"F0ERPLA"	Q 600.4	BOOL	// [F0IM1.F0S11]: F0: EV RECUO PILOTO A
"F0ERSRB"	Q 600.5	BOOL	// [F0IM1.F0S11]: F0: EV RECUO SERRAGE B
"F0IM_F0S11_R1"	Q 600.6	BOOL	// [F0IM1.F0S11]: RESERVA
"F0ERSRD"	Q 600.7	BOOL	// [F0IM1.F0S11]: F0: EV RECUO SERRAGE D
"F0ERRCE"	Q 601.0	BOOL	// [F0IM1.F0S12]: F0: EV RECUO RETACAGE E
"F0EACAF"	Q 601.1	BOOL	// [F0IM1.F0S12]: F0: EV AVANÇO CARRO F
"F0EARCF1"	Q 601.2	BOOL	// [F0IM1.F0S12]: F0: EV AVANÇO RETACAGE F1
"F0IM_F0S12_R1"	Q 601.3	BOOL	// [F0IM1.F0S12]: RESERVA
"F0EARCE"	Q 601.4	BOOL	// [F0IM1.F0S12]: F0: EV AVANÇO RETACAGE E
"F0ERCAF"	Q 601.5	BOOL	// [F0IM1.F0S12]: F0: EV RECUO CARRO F
"F0IM_F0S12_R2"	Q 601.6	BOOL	// [F0IM1.F0S12]: RESERVA
"F0IM_F0S12_R3"	Q 601.7	BOOL	// [F0IM1.F0S12]: RESERVA
"G0EAPLA"	Q 620.0	BOOL	// [G0IM1.G0S11]: G0: EV AVANÇO PILOTO A
"G0EASRB"	Q 620.1	BOOL	// [G0IM1.G0S11]: G0: EV AVANÇO SERRAGE B
"G0IM_G0S13_R1"	Q 620.2	BOOL	// [G0IM1.G0S11]: RESERVA
"G0IM_G0S13_R2"	Q 620.3	BOOL	// [G0IM1.G0S11]: RESERVA
"G0ERPLA"	Q 620.4	BOOL	// [G0IM1.G0S11]: G0: EV RECUO PILOTO A
"G0ERSRB"	Q 620.5	BOOL	// [G0IM1.G0S11]: G0: EV RECUO SERRAGE B
"G0IM_G0S13_R3"	Q 620.6	BOOL	// [G0IM1.G0S11]: RESERVA
"G0IM_G0S13_R4"	Q 620.7	BOOL	// [G0IM1.G0S11]: RESERVA
"RESERVA-"	Q 640.7	BOOL	// [H0IM1.H0S11]: H0: RESERVA
"K0EASR1"	Q 650.0	BOOL	// [K0TDS1] K0: EV AVANCE SR1
"K0ERSR1"	Q 650.1	BOOL	// [K0TDS1] K0: EV RETROCESO SR1
"K0EASR2"	Q 650.2	BOOL	// [K0TDS1] K0: EV AVANCE SR2
"K0ERSR2"	Q 650.3	BOOL	// [K0TDS1] K0: EV RETROCESO SR2
"K0S11_RESERVA1"	Q 650.4	BOOL
"K0S11_RESERVA2"	Q 650.5	BOOL
"K0EASR3"	Q 650.6	BOOL	// [K0TDS1] K0: EV AVANCE SR3
"K0ERSR3"	Q 650.7	BOOL	// [K0TDS1] K0: EV RETROCESO SR3
"K0_VVAL"	Q 656.0	BOOL	// [K0A2] Habilitacion de 24V Valvulas CPX K0TDS1
"K0EVCPX"	Q 656.1	BOOL	// [K0A2] ELECTROVÁLVULA CPX K0TDS1
"Z2RCM"	Q 800.7	BOOL	// [Z2ZB.M05]: Z2 GROUND CONTROL RELAY
"Z2RSC1"	Q 815.0	BOOL	// [Z2ZB.M09]: RELAY SAFETY COMMON 1 (AU)
"Z2RES"	Q 815.1	BOOL	// [Z2ZB.M09]: RELAY SAFETY COMMON 2 (ES)
"Z2RFZ"	Q 815.2	BOOL	// [Z2ZB.M09]: RELAY SAFETY COMMON 3 (RFZ)
"Z2RSC4"	Q 815.3	BOOL	// [Z2ZB.M09]: RELAY SAFETY COMMON 4 (SC4)
"B1OP1VAT"	Q 821.0	BOOL	// B1 Lampara autorizacion de trabajo
"B1OP1VIT"	Q 821.1	BOOL	// B1 Lampara de prohibicion de trabajo
"B1OP1VDF"	Q 821.2	BOOL	// B1 Lampara de defecto
"B0RFRO1"	Q 841.0	BOOL	// [B0SB.M11]: B0 SAFETY COMMON 3 (FRO1)
"B0RFRO2"	Q 841.1	BOOL	// [B0SB.M11]: B0 SAFETY COMMON 4 (FRO2)
"B0RFRO3"	Q 841.2	BOOL	// [B0SB.M11]: B0 SAFETY COMMON 5 (FRO3)
"C1OP1VAT"	Q 851.0	BOOL	// C1 Lampara autorizacion de trabajo
"C1OP1VIT"	Q 851.1	BOOL	// C1 Lampara de prohibicion de trabajo
"C1OP1VDF"	Q 851.2	BOOL	// C1 Lampara de defecto
"C0RFRO1"	Q 871.0	BOOL	// [C0SB.M11]: C0 SAFETY COMMON 3 (C0SOP)
"C0RFRO2"	Q 871.1	BOOL	// [C0SB.M11]: C0 SAFETY COMMON 4 (C0)
"C0RFRO3"	Q 871.2	BOOL	// [C0SB.M11]: C0 SAFETY COMMON 5 (C0)
"E1OP1VAT"	Q 881.0	BOOL	// E1 Lampara autorizacion de trabajo
"E1OP1VIT"	Q 881.1	BOOL	// E1 Lampara de prohibicion de trabajo
"E1OP1VDF"	Q 881.2	BOOL	// E1 Lampara de defecto
"E2OP2VAT"	Q 881.5	BOOL
"E2OP2VIT"	Q 881.6	BOOL
"E0RFRO1"	Q 901.0	BOOL	// [E0SB.M11]: E0 SAFETY COMMON 3 ( E0SOP)
"E0RFRO2"	Q 901.1	BOOL	// [E0SB.M11]: E0 SAFETY COMMON 4 ( E0)
"E0RFRO3"	Q 901.2	BOOL	// [E0SB.M11]: E0 SAFETY COMMON 5 ( E0)
"G1OP1VAT"	Q 911.0	BOOL	// B1 Lampara autorizacion de trabajo
"G1OP1VIT"	Q 911.1	BOOL	// B1 Lampara de prohibicion de trabajo
"G1OP1VDF"	Q 911.2	BOOL	// B1 Lampara de defecto
"G0RFRO1"	Q 931.0	BOOL	// [G0SB.M11]: G0 SAFETY COMMON 3 (G0SOP)
"G0RFRO2"	Q 931.1	BOOL	// [G0SB.M11]: G0 SAFETY COMMON 4 (G0)
"G0RFRO3"	Q 931.2	BOOL	// [G0SB.M11]: G0 SAFETY COMMON 5 (G0)
"J1OP1VAT"	Q 940.0	BOOL	// J1 Lampara autorizacion de trabajo
"J1OP1VIT"	Q 940.1	BOOL	// J1 Lampara de prohibicion de trabajo
"J1OP1VDF"	Q 940.2	BOOL	// J1 Lampara de defecto
"B0EAPL1"	Q 950.0	BOOL	// [B0DTS1]: B0: EV AVANCE PL1
"B0ERPL1"	Q 950.1	BOOL	// [B0DTS1]: B0: EV RETROCESO PL1
"B0EASR2"	Q 950.2	BOOL	// [B0DTS1]: B0: EV AVANCE SR2
"B0ERSR2"	Q 950.3	BOOL	// [B0DTS1]: B0: EV RETROCESO SR2
"B0EASR3"	Q 950.4	BOOL	// [B0DTS1]: B0: EV AVANCE SR3
"B0ERSR3"	Q 950.5	BOOL	// [B0DTS1]: B0: EV RETROCESO SR3
"C0EAPL1"	Q 960.0	BOOL	// [C0DTS1]: C0: EV AVANCE PL1
"C0ERPL1"	Q 960.1	BOOL	// [C0DTS1]: C0: EV RETROCESO PL1
"C0EASR2"	Q 961.2	BOOL	// [C0DTS1]: C0: EV AVANCE SR2
"C0ERSR2"	Q 961.3	BOOL	// [C0DTS1]: C0: EV RETROCESO SR2
"C0EASR3"	Q 961.4	BOOL	// [C0DTS1]: C0: EV AVANCE SR3
"C0ERSR3"	Q 961.5	BOOL	// [C0DTS1]: C0: EV RETROCESO SR3
"E0EASR1"	Q 1040.0	BOOL	// [E0TDS1]: E0: EV AVANCE SR1
"E0ERSR1"	Q 1040.1	BOOL	// [E0TDS1]: E0: EV RETROCESO SR1
"E0EASR2"	Q 1040.2	BOOL	// [E0TDS1]: E0: EV AVANCE SR2
"E0ERSR2"	Q 1040.3	BOOL	// [E0TDS1]: E0: EV RETROCESO SR2
"E0EASR3"	Q 1040.4	BOOL	// [E0TDS1]: E0: EV AVANCE SR3
"E0ERSR3"	Q 1040.5	BOOL	// [E0TDS1]: E0: EV RETROCESO SR3
"E0EAVU4"	Q 1040.6	BOOL	// [E0TDS1]: E0: EV AVANCE VU4
"E0ERVU4"	Q 1040.7	BOOL	// [E0TDS1]: E0: EV RETROCESO VU4
"E0EAVU5"	Q 1041.0	BOOL	// [E0TDS1]: E0: EV AVANCE VU5
"E0ERVU5"	Q 1041.1	BOOL	// [E0TDS1]: E0: EV RETROCESO VU5
"E0EASR6"	Q 1041.2	BOOL	// [E0TDS1]: E0: EV AVANCE SR6
"E0ERSR6"	Q 1041.3	BOOL	// [E0TDS1]: E0: EV RETROCESO SR6
"G0EASR1"	Q 1060.0	BOOL	// [G0TDS1]: G0: EV AVANCE SR1
"G0ERSR1"	Q 1060.1	BOOL	// [G0TDS1]: G0: EV RETROCESO SR1
"G0EASR2"	Q 1060.2	BOOL	// [G0TDS1]: G0: EV AVANCE SR2
"G0ERSR2"	Q 1060.3	BOOL	// [G0TDS1]: G0: EV RETROCESO SR2
"G0EASR3"	Q 1060.4	BOOL	// [G0TDS1]: G0: EV AVANCE SR3
"G0ERSR3"	Q 1060.5	BOOL	// [G0TDS1]: G0: EV RETROCESO SR3
"L1VROC"	Q 1070.0	BOOL	// L1: LED BOTON RETORNO A ORIGEN
"L1VIT"	Q 1070.2	BOOL	// L1: LAMPARA DE PROHIBICION DE TRABAJO
"L1VDF"	Q 1070.3	BOOL	// L1: LAMPARA DE DEFECTO
"L1VAT"	Q 1070.4	BOOL	// L1: LAMPARA DE PROHIBICION DE TRABAJO
"L0EAPS1"	Q 1071.0	BOOL	// L0: Electrovalvula de avance PIN SHIFT 1
"L0ERPS1"	Q 1071.1	BOOL	// L0: Electrovalvula de retroceso PIN SHIFT 1
"L0EASR1"	Q 1071.2	BOOL	// L0: Electrovalvula de avance CLAMP 1
"L0ERSR1"	Q 1071.3	BOOL	// L0: Electrovalvula de retroceso CLAMP 1
"L0EASR2"	Q 1071.4	BOOL	// L0: Electrovalvula de avance CLAMP 2
"L0ERSR2"	Q 1071.5	BOOL	// L0: Electrovalvula de retroceso CLAMP 2
"L0EASR3"	Q 1071.6	BOOL	// L0: Electrovalvula de avance CLAMP 3
"L0ERSR3"	Q 1071.7	BOOL	// L0: Electrovalvula de retroceso CLAMP 3
"L0EAVU1"	Q 1072.0	BOOL	// L0: Electrovalvula de avance EJECTOR 1
"L0ERVU1"	Q 1072.1	BOOL	// L0: Electrovalvula de retroceso EJECTOR 1
"L0EAVU2"	Q 1072.2	BOOL	// L0: Electrovalvula de avance PINGYI 1
"L0ERVU2"	Q 1072.3	BOOL	// L0: Electrovalvula de retroceso PINGYI 1
"L0EASR4"	Q 1072.4	BOOL	// L0: ELECTROVALVULA DE AVANCE MOV SR4 (DETECTOR DPP15)
"L0ERSR4"	Q 1072.5	BOOL	// L0: ELECTROVALVULA DE AVANCE MOV SR4 (DETECTOR DPP15)
"FDIS_90_8_AckCan"	Q 1080.0	BOOL	// FESTO DI-Safe error de canal 90 - 8 L0
"FDIS_90_8_Pass"	Q 1080.1	BOOL	// FESTO DI-Safe 90 - 8 1 PASSIVATION PAR CANAL / 0 - PASSIVATION PAR MODULE
"L0SOP"	Q 1087.0	BOOL
"L024SV"	Q 1087.1	BOOL	// L0 24V SUPPLY FOR SOFSTART VALVE
"M1VROC"	Q 1100.0	BOOL	// M1: LAMPARA DE RETORNO AL ORIGEN
"M1VIT"	Q 1100.2	BOOL	// M1: LAMPARA DE PROHIBICION DE TRABAJO
"M1VDF"	Q 1100.3	BOOL	// M1: LAMPARA DE DEFECTO
"M1VAT"	Q 1100.4	BOOL	// M1: LAMPARA DE PERMISO DE TRABAJO
"FDIS_100_5_AckCan"	Q 1104.0	BOOL	// FESTO DI-Safe ERROR DE CANAL M0
"FDIS_100_5_Pass"	Q 1104.1	BOOL	// FESTO DI-Safe 1 - passivation par canal / 0 - passivation par module
"M0SOP"	Q 1111.0	BOOL
"M024SV"	Q 1111.1	BOOL	// M0 24V SUPPLY FOR SOFSTART VALVE
"M0EASR1"	Q 1117.0	BOOL	// M0: Electrovalvula avance HAND CLAMP 1
"M0ERSR1"	Q 1117.1	BOOL	// M0: Electrovalvula retroceso HAND CLAMP 1
"M0EASR2"	Q 1117.2	BOOL	// M0: Electrovalvula avance CLAMP 1
"M0ERSR2"	Q 1117.3	BOOL	// M0: Electrovalvula retroceso CLAMP 1
"M0EAVU1"	Q 1117.4	BOOL	// M0: Electrovalvula avance EJECTOR 1
"M0ERVU1"	Q 1117.5	BOOL	// M0: Electrovalvula retroceso EJECTOR 1
"N0EAPLC"	Q 1150.4	BOOL
"N0ERPLC"	Q 1150.5	BOOL
"N0EASRD"	Q 1150.6	BOOL
"N0ERSRD"	Q 1150.7	BOOL
"N0EASRE"	Q 1151.0	BOOL
"N0ERSRE"	Q 1151.1	BOOL
"N0EASRF"	Q 1151.2	BOOL
"N0ERSRF"	Q 1151.3	BOOL
"N0EACLH"	Q 1151.6	BOOL
"N0ERCLH"	Q 1151.7	BOOL
"N0EASRJ"	Q 1152.0	BOOL
"N0ERSRJ"	Q 1152.1	BOOL
"N0EACLK"	Q 1152.2	BOOL
"N0ERCLK"	Q 1152.3	BOOL
"N0EBLK"	Q 1152.4	BOOL	// ElectroValvula Bloqueti Cilindro K
"N1VDF"	Q 1155.0	BOOL	// N1: LAMPARA DE DEFECTO
"N1VAT"	Q 1155.1	BOOL	// N1: LAMPARA DE PERMISO DE TRABAJO
"N1VIT"	Q 1155.3	BOOL	// N1: LAMPARA DE PROHIBICION DE TRABAJO
"N0EAPLA"	Q 1156.0	BOOL
"N0ERPLA"	Q 1156.1	BOOL
"N0EACLB"	Q 1156.2	BOOL
"N0ERCLB"	Q 1156.3	BOOL
"N0EACLG"	Q 1156.4	BOOL
"N0ERCLG"	Q 1156.5	BOOL
"FDIS_110_5_AckCan"	Q 1158.0	BOOL	// FESTO DI-Safe ERROR DE CANAL M0
"FDIS_110_5_Pass"	Q 1158.1	BOOL	// FESTO DI-Safe 1 - passivation par canal / 0 - passivation par modul
"N0SOP"	Q 1165.0	BOOL	// N0IM1: COMUN SEGURIDAD OPERADO
"N0EVAIR"	Q 1165.1	BOOL	// N0 ELECTROVALVULA DE AIRE GENERAL
"FDIS_90_8_M"	QW 1081	INT	// FESTO DI-Safe 90-8 MODE L0
"FDIS_100_5_M"	QW 1105	INT	// FESTO DI-Safe 100 - 5 MODE
"FDIS_110_5_M"	QW 1159	INT	// FESTO DI-Safe 110 - 5 MODE
"TP"	SFB 3	SFB 3	// GENERATE A PULSE
"TON"	SFB 4	SFB 4	// GENERATE AN ON DELAY
"TOF"	SFB 5	SFB 5	// GENERATE AN OFF DELAY
"RDREC"	SFB 52	SFB 52	// READ A PROCESS DATA RECORD
"WRREC"	SFB 53	SFB 53	// WRITE A PROCESS DATA RECORD
"RALRM"	SFB 54	SFB 54	// Receive Alarm Data
"SET_CLK"	SFC 0	SFC 0	// SET SYSTEM CLOCK
"READ_CLK"	SFC 1	SFC 1	// READ SYSTEM CLOCK
"RD_SINFO"	SFC 6	SFC 6	// READ OB START INFORMATION
"D_ACT_DP"	SFC 12	SFC 12	// DEACTIVATING AND ACTIVATING DP SLAVES
"DPRD_DAT"	SFC 14	SFC 14	// READ CONSISTENT DATA OF A STANDARD DP SLAVE
"DPWR_DAT"	SFC 15	SFC 15	// WRITE CONSISTENT DATA TO A STANDARD DP SLAVE
"BLKMOV"	SFC 20	SFC 20	// COPY VARIABLES
"FILL"	SFC 21	SFC 21	// INITIALIZE A MEMORY AREA
"TEST_DB"	SFC 24	SFC 24	// TEST DATA BLOCK
"DIS_AIRT"	SFC 41	SFC 41	// DELAY THE HIGHER PRIORITY INTERRUPTS AND ASYNCHRONOUS ERRORS
"EN_AIRT"	SFC 42	SFC 42	// ENABLE HIGHER PRIORITY INTERRUPTS AND ASYNCHRONOUS ERRORS
"STP"	SFC 46	SFC 46	// CHANGE THE CPU TO STOP
"RDSYSST"	SFC 51	SFC 51	// READ A SYSTEM STATUS LIST OR PARTIAL LIST
"WR_REC"	SFC 58	SFC 58	// WRITE DATA RECORD
"RD_REC"	SFC 59	SFC 59	// READ A DATA RECORD
"TIME_TCK"	SFC 64	SFC 64	// READ THE SYSTEM TIME
"GEO_LOG"	SFC 70	SFC 70	// DETERMINE LOGICAL ADDRESS
"READ_DBL"	SFC 83	SFC 83	// READ DATA BLOCK OUT OF LOAD MEMORY
"WRIT_DBL"	SFC 84	SFC 84	// WRITE DATA BLOCK IN LOAD MEMORY
"DEL_SI"	SFC 106	SFC 106	// Deleting Dynamically Assigned System Instances
"ALARM_DQ"	SFC 107	SFC 107	// Creating Acknowledgeable Block-related Message
"ALARM_D"	SFC 108	SFC 108	// Creating Acknowledged Block-related Message
"LIEN_SEC"	UDT 1507	UDT 1507	// TABLE COMMUNE AUX BF_ZONE_PORTE1, BF_ZONE_RSEC1, BF_ZONE_MODE_IHM, BF_ZONE_AIR
"MOT_FONC_DPL"	UDT 1866	UDT 1866
"LIEN_PUP"	UDT 1988	UDT 1988	// Gestion des Modes et des pupitres de cde manu de la  zone (BF_ZONE_MODE_IHM)
"LIEN_ILOT"	UDT 2004	UDT 2004	// INFO CONTROL LINKED TO THE FACILITY (BF_ILOT)
"MOT_FONC_MP"	UDT 2041	UDT 2041	// INFO CONTROL OF A MOVEMENT (BF_MOUVMP1)
"MOT_FONC"	UDT 2042	UDT 2042	// INFO D'UN MOUVEMENT (BF_MOUV2P1,BF_MVSE2P1, BF_RB_COD_PREH_API)
"VAT_SIPTOL"	VAT 1	
"VAT_TALOA0"	VAT 2	
"VAT_BASE DE DADOS"	VAT 3	
"Z1T_TEMPOS"	VAT 4	
"Z2T_TEMPOS"	VAT 5	
"VAT_6"	VAT 6	
"acompanhamento zona 8"	VAT 7		// teste tucker
"TOMAS"	VAT 8	
"W0"	VAT 9	
"VAT_Z1_BOT_EMER"	VAT 10	
"VAT_Z2_BOT_EMER"	VAT 11		// BOTAO_DE_EMERGENCIA
"VAT_Z1_VALIDAÇÃO"	VAT 12	
"VAT_CDIV_2"	VAT 13	
"VAT_Z2_VALIDAÇÃO"	VAT 14	
"ELEV_CARREGAMENTO"	VAT 15	
"ELEV_DESCARREGAMENTO"	VAT 16	
"VAT_17"	VAT 17	
"TESTE_MODO_DEGR"	VAT 18	
"Z2_SIPTOL"	VAT 19	
"mostrar IIT"	VAT 20	
"tab_iit_2"	VAT 21	
"VAT_22"	VAT 22	
"afficher"	VAT 23	
"VAT_24"	VAT 24	
"SIPTOL_X52_X67_X60"	VAT 25	
"Z3_SIPTOL"	VAT 26		// VAT SIPTOL ZONA 3
"VAT_IIT"	VAT 27	
"VAT_Z1T"	VAT 28	
"SMP"	VAT 29	
"def_qbad"	VAT 30	
END_SYMBOL_TABLE

SYMBOL_TABLE
"CC1"	C 1	COUNTER	// Contador Cabeçote 1
"CC2"	C 2	COUNTER	// Contador Cabeçote 2
"CC3"	C 3	COUNTER	// Contador Cabeçote 3
"CT_M6_FAG0014"	C 4	COUNTER	// Contador de tucker pistola 1 do DCE FAG0014
"CT_M6_FAG0039"	C 5	COUNTER	// Contador de tucker pistola 3 do DCE FAG0039
"CT_P1M6_RF60"	C 6	COUNTER	// CONTADOR PISTOLA 1 M6 RF60
"CT_P2M6_RF60"	C 7	COUNTER	// CONTADOR PISTOLA 2 M6 RF60
"I01"	DB 1	FB 1	// FACILITY: INSTANCE DB (FB1)
"I02"	DB 2	FB 2	// FACILITY: INSTANCE DB FOR MMC CONTROL (FB2)
"I03"	DB 3	FB 3	// FACILITY: INSTANCE DB FOR MOP/LOP
"I04"	DB 4	FB 4
"CDIV"	DB 69	DB 69	// FACILITY: DIVERSITIES CODES TABLE / TABLE CODES DIVERSITES
"SFM_DB"	DB 75	FB 20	// FACILITY: DB FAILURE MESSAGE (SFM_FB) LINK WITH PROFINET CONTROL
"SFM_GLOBAL_DB"	DB 76	DB 76	// DIAGNOSTIC BLOCK FOR THE SIGNALISATION OF THE SYSTEM ERRORS
"SFM_PN"	DB 77	DB 77	// PROFINET DIAGNOSTIC FUNCTION EDITING DB FOR IHMP
"SIP1"	DB 89	DB 89	// SIPTOL EXCHANGES DATAS / TABLE D'ECHANGES SIPTOL
"PILE"	DB 90	DB 90	// FACILITY: FIFO STORAGE / PILE DE STOCKAGE
"CAB"	DB 91	DB 91	// L0: BARCODE READER DB / DB LECTEUR CODE BARRE
"IDENT"	DB 93	DB 93	// RFID DATAS / IDENTIFIANT DYNAMIQUE
"IBD"	DB 95	DB 95	// FACILITY: DATA BASE DB / DB BASE DE DONNEE
"IIT"	DB 96	DB 96	// FACILITY: PART TABLE / DB TABLE PIECE
"IG"	DB 99	DB 99	// FACILITY: GLOBAL DB / DB GLOBAL
"Z1"	DB 100	FB 100	// ZONE 1: INSTANCE DB
"Z1A0"	DB 110	FB 110	// A0 MONTAGE INSTANCE DATA BLOC / BLOC DE DONNEES INSTANCE A0 MONTAGE
"Z1A1"	DB 111	FB 111	// A1 OP_BIMA INSTANCE DATA BLOC / BLOC DE DONNEES INSTANCE A1 OP_BIMA
"Z1A2"	DB 112	FB 112	// A2 OP_BIMA INSTANCE DATA BLOC / BLOC DE DONNEES INSTANCE A2 OP_BIMA
"Z1A0L"	DB 114	FB 114	// A0 LANCEMENT INSTANCE DATA BLOC / BLOC DE DONNEES INSTANCE A0 LANCEMENT
"Z1D0"	DB 140	FB 140	// D0 MONTAGE INSTANCE DATA BLOC / BLOC DE DONNEES INSTANCE D0 MONTAGE
"Z1D1"	DB 141	FB 141	// D1 OP_BIMA INSTANCE DATA BLOC / BLOC DE DONNEES INSTANCE D1 OP_BIMA
"Z1D2"	DB 142	FB 142	// D2 OP_BIMA INSTANCE DATA BLOC / BLOC DE DONNEES INSTANCE D2 OP_BIMA
"Z1F0"	DB 150	FB 150	// F0 MONTAGE INSTANCE DATA BLOC / BLOC DE DONNEES INSTANCE F0 MONTAGE
"Z1F1"	DB 151	FB 151	// F1 OP_BIMA INSTANCE DATA BLOC / BLOC DE DONNEES INSTANCE F1 OP_BIMA
"Z1F2"	DB 152	FB 152	// F2 OP_BIMA INSTANCE DATA BLOC / BLOC DE DONNEES INSTANCE F2 OP_BIMA
"Z1F3"	DB 153	FB 253	// F3 OP_BIMA INSTANCE DATA BLOC / BLOC DE DONNEES INSTANCE F3 OP_BIMA
"Z1N0"	DB 160	FB 160
"Z1N1"	DB 161	FB 161
"Z1K0"	DB 170	FB 170
"Z1K1"	DB 171	FB 171
"Z1T"	DB 198	DB 198	// ZONE 1: REFERENCE TIME FOR MOVEMENTS
"Z1G"	DB 199	DB 199	// ZONE 1: GLOBAL DB
"Z2"	DB 200	FB 200	// ZONE 2: INSTANCE DB
"Z2B0"	DB 210	FB 210
"Z2B1"	DB 211	FB 211
"Z2C0"	DB 240	FB 240
"Z2C1"	DB 241	FB 241
"Z2C2"	DB 242	FB 242
"Z2E0"	DB 250	FB 250
"Z2E1"	DB 251	FB 251
"Z2E2"	DB 252	FB 252	// E2 OP_BIMA INSTANCE DATA BLOC / BLOC DE DONNEES INSTANCE E2 OP_BIMA
"Z2E0L"	DB 254	FB 254
"Z2G0"	DB 260	FB 260
"Z2G1"	DB 261	FB 261
"Z2G2"	DB 262	FB 262
"Z2J0"	DB 270	FB 270
"Z2T"	DB 298	DB 298	// ZONE 2: REFERENCE TIME FOR MOVEMENTS
"Z2G"	DB 299	DB 299	// ZONE 2: GLOBAL DB
"Z3"	DB 300	FB 300
"Z3L0"	DB 310	FB 310
"Z3L1"	DB 311	FB 311
"Z3L2"	DB 312	FB 312
"Z3L0L"	DB 313	FB 313
"Z3M0"	DB 320	FB 320
"Z3M1"	DB 321	FB 321
"Z3M2"	DB 322	FB 322
"Z3T"	DB 398	DB 398
"Z3G"	DB 399	DB 399
"Z8"	DB 800	FB 800	// ZONE 8: INSTANCE DB
"Z8X0"	DB 810	FB 810	// X0 CHAINE INSTANCE DATA BLOC / BLOC DE DONNEES INSTANCE X0 CHAINE
"Z8X1"	DB 811	FB 811	// X1 OP_BPVAL INSTANCE DATA BLOC / BLOC DE DONNEES INSTANCE X1 OP_BPVAL
"Z8W0"	DB 815	FB 815
"Z8Y0"	DB 820	FB 820	// Y0 CHAINE INSTANCE DATA BLOC / BLOC DE DONNEES INSTANCE Y0 CHAINE
"Z8Y1"	DB 821	FB 821	// Y1 OP_BPVAL INSTANCE DATA BLOC / BLOC DE DONNEES INSTANCE Y1 OP_BPVAL
"Z8T"	DB 898	DB 898	// ZONE 8: REFERENCE TIME FOR MOVEMENTS
"Z8G"	DB 899	DB 899	// ZONE 8: GLOBAL DB
"A0BARCODE"	DB 900	DB 900	// DADOS DO BARCODE A SER CARREGADOS NA TALO
"A0TALO"	DB 951	DB 951	// A0: LOCAL TABLE / TABLE LOCALE
"A0wTALO"	DB 952	DB 952	// A0w: LOCAL TABLE / TABLE LOCALE
"B0TALO"	DB 953	DB 953	// B0: LOCAL TABLE / TABLE LOCALE
"B0wTALO"	DB 954	DB 954	// B0w: LOCAL TABLE / TABLE LOCALE
"C0TALO"	DB 955	DB 955	// C0: LOCAL TABLE / TABLE LOCALE
"C0wTALO"	DB 956	DB 956	// C0w: LOCAL TABLE / TABLE LOCALE
"D0TALO"	DB 957	DB 957	// D0: LOCAL TABLE / TABLE LOCALE
"D0wTALO"	DB 958	DB 958	// D0w: LOCAL TABLE / TABLE LOCALE
"E0TALO"	DB 959	DB 959	// E0: LOCAL TABLE / TABLE LOCALE
"E0wTALO"	DB 960	DB 960	// E0w: LOCAL TABLE / TABLE LOCALE
"F0TALO"	DB 961	DB 961	// F0: LOCAL TABLE / TABLE LOCALE
"F0wTALO"	DB 962	DB 962	// F0w: LOCAL TABLE / TABLE LOCALE
"G0TALO"	DB 963	DB 963	// G0: LOCAL TABLE / TABLE LOCALE
"G0wTALO"	DB 964	DB 964	// G0w: LOCAL TABLE / TABLE LOCALE
"TRM"	DB 1098	DB 1098	// FACILITY: SAFETY OPERATOR CONTROL
"ITS0"	DB 1100	FB 1100	// FACILITY: SAFETY CONTROL DB
"ITSZ1_AU_ES_FZ"	DB 1110	FB 1110	// ZONE 1: SAFETY CONTROL INSTANCE DB (AU ES FZ)
"ITSZ1_SOP"	DB 1111	FB 1111	// ZONE 1: SAFETY CONTROL INSTANCE DB (SOP)
"ITSZ2_AU_ES_FZ"	DB 1120	FB 1120	// ZONE 2: SAFETY CONTROL INSTANCE DB (AU ES FZ)
"ITSZ2_SOP"	DB 1121	FB 1121	// ZONE 2: SAFETY CONTROL INSTANCE DB (SOP)
"ITSZ2VAR"	DB 1123	FB 1123	// Z2 : DB D'INSTANCE DU FB 1123
"ITSZ3_AU_ES_FZ"	DB 1130	FB 1130
"ITSZ3_SOP"	DB 1131	FB 1131
"ITSZ8_AU_ES_FZ"	DB 1180	FB 1180	// ZONE 1: SAFETY CONTROL INSTANCE DB EMERGENCY STOP (AU)
"ITSZ8_SOP"	DB 1181	FB 1181	// ZONE 1: SAFETY CONTROL INSTANCE DB STARTING-UP (ES)
"ITSZ8_RLV"	DB 1182	FB 1182	// Z8 : DB D'INSTANCE DU FB 1182
"TSM"	DB 1279	DB 1279	// FACILITY: SAFETY CONTROL DB
"F_GLOBDB"	DB 1300	DB 1300
"F01165_N0FS3"	DB 1301	FB 1300
"F01158_N0FE5"	DB 1302	FB 1300
"F00913__G0SB___M08"	DB 1303	FB 1300
"F00919__G0SB___M09"	DB 1304	FB 1300
"F00925__G0SB___M10"	DB 1305	FB 1300
"F00931__G0SB___M11"	DB 1306	FB 1300
"F00883__E0SB___M08"	DB 1307	FB 1300
"F00889__E0SB___M09"	DB 1308	FB 1300
"F00895__E0SB___M10"	DB 1309	FB 1300
"F00901__E0SB___M11"	DB 1310	FB 1300
"F00853__C0SB___M08"	DB 1311	FB 1300
"F00859__C0SB___M09"	DB 1312	FB 1300
"F00865__C0SB___M10"	DB 1313	FB 1300
"F00871__C0SB___M11"	DB 1314	FB 1300
"F00841__B0SB___M11"	DB 1315	FB 1300
"F00835__B0SB___M10"	DB 1316	FB 1300
"F00829__B0SB___M09"	DB 1317	FB 1300
"F00823__B0SB___M08"	DB 1318	FB 1300
"F00815__Z2ZB___M09"	DB 1319	FB 1300
"F00809__Z2ZB___M08"	DB 1320	FB 1300
"F00803__Z2ZB___M07"	DB 1321	FB 1300
"F00290__F0SB___M11"	DB 1322	FB 1300
"F00284__F0SB___M10"	DB 1323	FB 1300
"F00278__F0SB___M09"	DB 1324	FB 1300
"F00272__F0SB___M08"	DB 1325	FB 1300
"F00210__D0SB___M11"	DB 1326	FB 1300
"F00204__D0SB___M10"	DB 1327	FB 1300
"F00198__D0SB___M09"	DB 1328	FB 1300
"F00192__D0SB___M08"	DB 1329	FB 1300
"F00090__A0SB___M11"	DB 1330	FB 1300
"F00084__A0SB___M10"	DB 1331	FB 1300
"F00078__A0SB___M09"	DB 1332	FB 1300
"F00072__A0SB___M08"	DB 1333	FB 1300
"F00018__Z1ZB___M07"	DB 1334	FB 1300
"F00012__Z1ZB___M06"	DB 1335	FB 1300
"F00394__KOSB___M10"	DB 1336	FB 1300
"F00388__KOSB___M09"	DB 1337	FB 1300
"F00400__K0SB___M11"	DB 1338	FB 1300
"F00382__KOSB___M08"	DB 1339	FB 1300
"F00047__Z3ZB_M09"	DB 1340	FB 1300
"F00041__Z3ZB_M08"	DB 1341	FB 1300
"F00035__Z3ZB_M07"	DB 1342	FB 1300
"F01080_L0FE11"	DB 1343	FB 1300
"F01087_L0FS11"	DB 1344	FB 1300
"F01104_M0FE11"	DB 1345	FB 1300
"F01111_M0FS11"	DB 1346	FB 1300
"F00656_K0A2"	DB 1361	FB 1300
"FESTO-DI-SAFE-DB"	DB 1723	FB 1723
"AFF"	DB 1863	DB 1863	// SIEBERT DISPLAY STRING STORAGE / STOCKAGE MESSAGE AFFICHEUR SIEBERT
"DB_IHM_WINCC"	DB 1962	FB 1962	// FACILITY: HMI INTERFACING WINCCFLEXIBLE RT
"DB_MMC"	DB 2000	DB 2000	// BACKUP COPY AND RESTORE OF EXTERN MEMORY MAP (MMC)
"DB_PN"	DB 2036	FB 2036	// INSTANCE IO PROFINET DB
"DB_PY"	DB 2222	FB 2222	// DB INSTANCE FB2222
"0_01_ILOT"	FB 1	FB 1	// FACILITY: FACILITY MANAGEMENT
"0_02_MMC"	FB 2	FB 2	// FACILITY: BACKUP MANAGEMENT AND DATA RESTITUTION ON EXTERNAL MMC CARD
"0_03_XOP"	FB 3	FB 3	// FACILITY: MOP/LOP MANAGEMENT
"0_04_COM"	FB 4	FB 4	// FACILITY: COM CONTROL WITH SIPTOL / GESTION DE LA COMMUNICATION AVEC SIPTOL
"SFM_FB"	FB 20	FB 20	// DIAGNOSTIC BLOCK FOR SYSTEM ERRORS SIGNALLING
"1_00_ZONE1"	FB 100	FB 100	// ZONE 1: ZONE CONTROL
"1_A0_MONTAGE"	FB 110	FB 110	// A0 MONTAGE FUNCTION BLOC / SECTION PROGRAMME A0 MONTAGE
"1_A1_OP_BIMA"	FB 111	FB 111	// A1 OP_BIMA FUNCTION BLOC / SECTION PROGRAMME A1 OP_BIMA
"1_A2_OP_BIMA"	FB 112	FB 112	// A2 OP_BIMA FUNCTION BLOC / SECTION PROGRAMME A2 OP_BIMA
"1_A3_OP_BIMA"	FB 113	FB 113	// A3 OP_BIMA FUNCTION BLOC / SECTION PROGRAMME A3 OP_BIMA
"1_A0_LANCEMENT"	FB 114	FB 114	// A0 LANCEMENT FUNCTION BLOC / SECTION PROGRAMME A0 LANCEMENT
"1_D0_MONTAGE"	FB 140	FB 140	// D0 MONTAGE FUNCTION BLOC / SECTION PROGRAMME D0 MONTAGE
"1_D1_OP_BIMA"	FB 141	FB 141	// D1 OP_BIMA FUNCTION BLOC / SECTION PROGRAMME D1 OP_BIMA
"1_D2_OP_BIMA"	FB 142	FB 142	// D2 OP_BIMA FUNCTION BLOC / SECTION PROGRAMME D2 OP_BIMA
"1_D3_OP_BIMA"	FB 143	FB 143	// D3 OP_BIMA FUNCTION BLOC / SECTION PROGRAMME D3 OP_BIMA
"1_D4_OP_BIMA"	FB 144	FB 144	// D4 OP_BIMA FUNCTION BLOC / SECTION PROGRAMME D4 OP_BIMA
"1_F0_MONTAGE"	FB 150	FB 150	// F0 MONTAGE FUNCTION BLOC / SECTION PROGRAMME F0 MONTAGE
"1_F1_OP_BIMA"	FB 151	FB 151	// F1 OP_BIMA FUNCTION BLOC / SECTION PROGRAMME F1 OP_BIMA
"1_F2_OP_BIMA"	FB 152	FB 152	// F2 OP_BIMA FUNCTION BLOC / SECTION PROGRAMME F2 OP_BIMA
"1_F3_OP_BIMA"	FB 153	FB 153	// F3 OP_BIMA FUNCTION BLOC / SECTION PROGRAMME F3 OP_BIMA
"1_N0_MONTAGE"	FB 160	FB 160
"1_N1_OP_BIMA"	FB 161	FB 161	// N1 OP_BIMA FUNCTION BLOC / SECTION PROGRAMME H1 OP_BIMA
"1_K0_MONTAGE"	FB 170	FB 170	// K0 MONTAGE FUNCTION BLOC / SECTION PROGRAMME K0 MONTAGE
"1_K1_OP_BIMA"	FB 171	FB 171	// K1 OP_BIMA FUNCTION BLOC / SECTION PROGRAMME K1 OP_BIMA
"F_TON"	FB 185	FB 185	// F_: Timer Switch On Delay
"F_TOF"	FB 186	FB 186	// F_: Timer Switch Off Delay
"2_00_ZONE2"	FB 200	FB 200	// ZONE 2: ZONE CONTROL
"2_B0_MONTAGE"	FB 210	FB 210	// B0 MONTAGE FUNCTION BLOC / SECTION PROGRAMME B0 MONTAGE
"2_B1_OP_BIMA"	FB 211	FB 211	// B1 OP_BIMA FUNCTION BLOC / SECTION PROGRAMME B1 OP_BIMA
"2_B0_LANCEMENT"	FB 214	FB 214	// B0 LANCEMENT FUNCTION BLOC / SECTION PROGRAMME B0 LANCEMENT
"2_H0_TABLE_TRAVAIL"	FB 220	FB 220
"2_H1_OP_BIMA"	FB 221	FB 221
"2_C0_MONTAGE"	FB 240	FB 240	// C0 MONTAGE FUNCTION BLOC / SECTION PROGRAMME C0 MONTAGE
"2_C1_OP_BIMA"	FB 241	FB 241	// C1 OP_BIMA FUNCTION BLOC / SECTION PROGRAMME C1 OP_BIMA
"2_C2_OP_BIMA"	FB 242	FB 242	// C2 OP_BIMA FUNCTION BLOC / SECTION PROGRAMME C1 OP_BIMA
"2_E0_MONTAGE"	FB 250	FB 250	// E0 MONTAGE FUNCTION BLOC / SECTION PROGRAMME E0 MONTAGE
"2_E1_OP_BIMA"	FB 251	FB 251	// E1 OP_BIMA FUNCTION BLOC / SECTION PROGRAMME E1 OP_BIMA
"2_E2_OP_BIMA"	FB 252	FB 252
"2_E0_LANCEMENT"	FB 254	FB 254	// E0 LANCEMENT FUNCTION BLOC / SECTION PROGRAMME E0 LANCEMENT
"2_G0_MONTAGE"	FB 260	FB 260	// G0 MONTAGE FUNCTION BLOC / SECTION PROGRAMME G0 MONTAGE
"2_G1_OP_BIMA"	FB 261	FB 261	// G1 OP_BIMA FUNCTION BLOC / SECTION PROGRAMME G1 OP_BIMA
"2_G2_OP_BIMA"	FB 262	FB 262
"2_J0_MONTAGE"	FB 270	FB 270	// J0 MONTAGE FUNCTION BLOC / SECTION PROGRAMME J0 MONTAGE
"3_00_ZONE 3"	FB 300	FB 300
"3_L0_MONTAGE"	FB 310	FB 310
"3_L1_OP_BIMA"	FB 311	FB 311
"3_L2_OP_BIMA"	FB 312	FB 312
"3_L0_LANCEMENT"	FB 313	FB 313
"3_M0_MONTAGE"	FB 320	FB 320
"3_M1_OP_BIMA"	FB 321	FB 321
"3_M2_OP_BIMA"	FB 322	FB 322
"8_00_ZONE8"	FB 800	FB 800	// ZONE 1: ZONE CONTROL
"8_X0_CHAINE"	FB 810	FB 810	// X0: CHAINE FUNCTION BLOCK
"8_X1_OP_BPVAL"	FB 811	FB 811	// X1 OP_BPVAL FUNCTION BLOC / SECTION PROGRAMME X1 OP_BPVAL
"8_W0_BUTEE"	FB 815	FB 815
"8_Y0_CHAINE"	FB 820	FB 820	// Y0: CHAINE FUNCTION BLOCK
"8_Y1_OP_BPVAL"	FB 821	FB 821	// Y1 OP_BPVAL FUNCTION BLOC / SECTION PROGRAMME X2 OP_BPVAL
"TS0"	FB 1100	FB 1100	// FACILITY: SAFETY CONTROL FB
"CONFIG_FESTO"	FB 1101	FB 1101	// ILOT: FB Gestion CONFIG FESTO
"TSZ1_AU_ES_FZ"	FB 1110	FB 1110	// ZONE 1: SAFETY CONTROL INSTANCE DB EMERGENCY STOP (AU)
"TSZ1_SOP"	FB 1111	FB 1111	// ZONE 1: SAFETY CONTROL INSTANCE DB STARTING-UP (ES)
"TSZ2_AU_ES_FZ"	FB 1120	FB 1120	// ZONE 2: SAFETY CONTROL INSTANCE FB (AU ES FZ)
"TSZ2_SOP"	FB 1121	FB 1121	// ZONE 2: SAFETY CONTROL INSTANCE DB STARTING-UP (ES)
"TSZ2_VAR"	FB 1123	FB 1123
"TSZ3_AU_ES_FZ"	FB 1130	FB 1130	// ZONA 2: SAFETY CONTROL INSTANCE DB EMERGENCY STOP
"TSZ3_SOP"	FB 1131	FB 1131
"TSZ8_AU_ES_FZ"	FB 1180	FB 1180	// ZONE 8: SAFETY CONTROL INSTANCE DB EMERGENCY STOP (AU)
"TSZ8_SOP"	FB 1181	FB 1181	// ZONE 8: SAFETY CONTROL INSTANCE FB (SOP)
"TSZ8_RLV"	FB 1182	FB 1182	// Z8: INSTANCE FB FOR RLV CONTROL
"F_IO_CGP"	FB 1300	FB 1300
"F_CTRL_1"	FB 1301	FB 1301
"F_CTRL_2"	FB 1302	FB 1302
"FISHL_W"	FB 1303	FB 1303
"FITON"	FB 1304	FB 1304
"FITOF"	FB 1305	FB 1305
"FI2HAND"	FB 1306	FB 1306
"F_DIAG_N"	FB 1307	FB 1307
"FIACK_GL"	FB 1308	FB 1308
"BF_MID_DIV"	FB 1603	FB 1603
"TUSEND"	FB 1681	FB 1681	// Send Data via UDP
"TCON"	FB 1685	FB 1685	// Connect
"F_2HAND"	FB 1688	FB 1688
"F_ACK_GL"	FB 1695	FB 1695	// Acquittement global de toutes les périphéries F d'un groupe d'exécution F
"P_SEND"	FB 1698	FB 1698	// Send Data to CP340
"P_RCV"	FB 1699	FB 1699	// Receive Data from CP340
"BFS_BSEC1"	FB 1710	FB 1710
"BFS_BSECTR1"	FB 1711	FB 1711
"BFS_AIR1"	FB 1713	FB 1713
"BFS_CRM1"	FB 1714	FB 1714
"BFS_CR1"	FB 1715	FB 1715
"BFS_BIMA"	FB 1719	FB 1719
"BFS_Festo-DIS-457"	FB 1723	FB 1723
"BF_DEVERM"	FB 1803	FB 1803	// BF STAGE DRY RUN CONTROL / BF GESTION DEVERMINAGE POSTE
"BF_G120DS_V2"	FB 1853	FB 1853	// G120D DRIVE BOX CONTROL / GESTION COFFRET VAR G120D
"BF_G120S_V2"	FB 1854	FB 1854	// Funcao Inverso G120 ScubeV2
"BF_CARACT_SIEBERT"	FB 1856	FB 1856	// SIEBERT DISPLAY MESSAGE CONFIGURATION / MISE EN FORME MESSAGE AFFICHEUR SIEBERT
"BF_RECALAGE2"	FB 1857	FB 1857
"BF_LANCEMENT"	FB 1858	FB 1858	// GESTION LANCEMENT SIPTOL
"BF_AFF SIEBERT (2*13) PN"	FB 1860	FB 1860
"BF_WELDING_BOX"	FB 1868	FB 1868	// WELDING BOX CONTROL / GESTION DES COFFRETS PARAMETRES SOUDURE
"BF_CONF_MACHINE"	FB 1869	FB 1869	// GESTION BASE DE DONNEE CONFIGURATION MACHINE
"BF_CODE_PROCESS"	FB 1870	FB 1870	// GESTION BASE DE DONNEE CODE PROCESS
"BF_DATABASE3"	FB 1871	FB 1871	// DATABASE MANAGEMENT / GESTION BASE DE DONNEES
"BF_IHMMUT1"	FB 1874	FB 1874
"BF_IHMCAME_ROBOT1"	FB 1875	FB 1875	// BF gérant l'IHM du bon fonctionnement de la came robot
"BF_IHMCR1"	FB 1876	FB 1876	// BF gérant l'IHM d'un element de la boucle de securite
"BF_IHMCRM1"	FB 1877	FB 1877	// BF gérant l'IHM du relais de controçle raccordement de masse CRM
"BF_CABRS"	FB 1897	FB 1897	// Barcode Reader / Lecteur de code a barre
"BF_ELEVAT"	FB 1900	FB 1900	// FB ELEVATEUR
"BF_IHMPORTE1"	FB 1930	FB 1930	// BF gérant l'IHM de la porte
"BF_IHMAIR1"	FB 1931	FB 1931	// BF gérant l'IHM du panneau pneumatique
"BF_ZONE_MODE_IHM1"	FB 1932	FB 1932	// Safety_V2: Zone HMI Operating _modes management/Gestion IHM et mode de la zone
"BF_IHMCR"	FB 1941	FB 1941	// BF gérant l'IHM du relais non piloté par l'API mais controlé
"BF_IHMCRM"	FB 1942	FB 1942	// BF gérant l'IHM du relais de controçle raccordement de masse CRM
"BF_IHMBSEC"	FB 1944	FB 1944	// BF - ZONE : Diagnostic SAFETY BFS_BSEC
"BF_IHMAIR"	FB 1948	FB 1948	// BF - ZONE : Diagnostic du bloc BFS_IHMAIR
"BF_MODBUS_MASTER_CP340"	FB 1958	FB 1958	// Modbus Maitre sur CP 340 (liaison serie)
"BF_MODBUS_SLAVE_CP340"	FB 1959	FB 1959	// Modbus Esclave avec CP 340
"BF_MODBUS_TCPIP_MASTER"	FB 1960	FB 1960	// BF gerant le protocole MODBUS TCP/IP en tant que Client TCP et Maitre MODBUS
"BF_MODBUS_TCPIP_SLAVE"	FB 1961	FB 1961	// Esclave Modbus sur CP Ethernet
"BF_IHM_WINCC"	FB 1962	FB 1962	// BF- Gestion images WinCC Flexible
"BF_ZONE_MODE_IHM"	FB 1963	FB 1963	// Zone: Traitement des Modes et des pupitre de cde manu de la  zone
"BF_MMC"	FB 2000	FB 2000	// Sauvegarde et restitution mémoire sur carte mémoire externe (MMC)
"BF_ILOT"	FB 2004	FB 2004	// BF- Gestion info lié à l'installation ( Ilot )
"BF_B_VIEAPI"	FB 2006	FB 2006	// Contrôle de la communication entre deux automates en liaison
"BF_TCY_SUIV"	FB 2019	FB 2019
"BF_RUP_FLU"	FB 2020	FB 2020	// Suivi - Rupture de Flux
"BF_CPT_PIECE"	FB 2021	FB 2021	// BF- Compteur de pièce
"BF_MULTIPOS2"	FB 2025	FB 2025	// COMMANDE MOUVEMENT MANUT HORIZONTAL ET VERTICAL JUSQU'A 16 POSITIONS
"BF_API_MAITRE_CAL"	FB 2031	FB 2031	// Gestion du Dialogue API MAITRE CAL
"BF_ACT_DESACT"	FB 2033	FB 2033	// BF- Activation désactivation d'un IO DEVICE
"BF_DIAG_PROFINET"	FB 2036	FB 2036	// BF- Diagnostic PROFINET IO
"BF_TF_TP"	FB 2037	FB 2037	// Transfert de table de mémoires pièces
"BF_FIFO"	FB 2039	FB 2039
"BF_MVSE2P1"	FB 2040	FB 2040	// Gestion d'un mouvement simple effet 2 positions
"BF_MOUVMP1"	FB 2041	FB 2041	// Gestion d'un mouvement multi position
"BF_MOUV2P1"	FB 2042	FB 2042	// BF- GESTION D'UN MOUVEMENT A 2 POSITIONS
"BF_PY"	FB 2222	FB 2222	// BLOCO VERIFICAÇÃO POKAYOKE (SELETTRA)
"0_00_CYCLE_ILOT"	FC 1	FC 1	// FACILITY: CALL OF FACILITY FB
"0_11_SECU_FERMEE"	FC 11	FC 11	// COPY OF SAFETY INFORMATION ZONE 1 TO 9 FOR THE SAFETY CLOSED ZONE
"SFM_FC"	FC 22	FC 22	// BLOCK DIAGNOSTIC FOR ERROR REPORTING SYSTEM
"1_00_CYCLE_Z1"	FC 100	FC 100	// ZONE 1: CALL OF FB ZONE
"2_00_CYCLE_Z2"	FC 200	FC 200	// ZONE 2: CALL OF FB ZONE
"3_00_CYCLE_Z3"	FC 300	FC 300
"8_00_CYCLE_Z8"	FC 800	FC 800	// ZONE 8: CALL OF FB ZONE
"0_00_TSAFETY"	FC 1100	FC 1100	// STD - FACILITY: EXECUTION F GROUP ASSOCIATE TO OB32 (NORMAL TASK)
"0_00_TSCYCLE"	FC 1101	FC 1101	// CALL OPERATOR NOT IN ZONE FB LINKED IN FACILITY
"F_SHR_W"	FC 1688	FC 1688	// F_: Shift right WORD
"F_SHL_W"	FC 1689	FC 1689	// F_: Shift left WORD
"AG_SEND"	FC 1698	FC 1698	// AG SEND
"AG_RECV"	FC 1699	FC 1699	// AG RECEIVE
"BADI"	I 0.0	BOOL	// [MOP-IM.M02]: FACILITY FAULT RESET BUTTON
"BRI"	I 0.1	BOOL	// [MOP-IM.M02]: FACILITY CONTROL ON BUTTON
"Z1BMCY"	I 0.2	BOOL	// [MOP-IM.M02]: CYCLE START BUTTON
"Z1SMM"	I 0.3	BOOL	// [MOP-IM.M02]: MANUAL SELECTOR
"Z1SMA"	I 1.0	BOOL	// [MOP-IM.M03]: AUTO SELECTOR
"Z1BMR1"	I 1.1	BOOL	// [MOP-IM.M03]: RETURN BUTTON
"Z1BMA1"	I 1.2	BOOL	// [MOP-IM.M03]: ADVANCE BUTTON
"CLIMOK"	I 1.3	BOOL	// [MOP-IM.M03]: AIR CONDITIONNING (OPTION)
"MOP-IM_M04_R1"	I 2.0	BOOL	// [MOP-IM.M04]: RESERVA
"MOP-IM_M04_R2"	I 2.1	BOOL	// [MOP-IM.M04]: RESERVA
"MOP-IM_M04_R3"	I 2.2	BOOL	// [MOP-IM.M04]: RESERVA
"MOP-IM_M04_R4"	I 2.3	BOOL	// [MOP-IM.M04]: RESERVA
"MOP-IM_M05_R1"	I 3.0	BOOL	// [MOP-IM.M05]: RESERVA
"MOP-IM_M05_R2"	I 3.1	BOOL	// [MOP-IM.M05]: RESERVA
"MOP-IM_M05_R3"	I 3.2	BOOL	// [MOP-IM.M05]: RESERVA
"MOP-IM_M05_R4"	I 3.3	BOOL	// [MOP-IM.M05]: RESERVA
"MOP-IM_M06_R1"	I 4.0	BOOL	// [MOP-IM.M06]: RESERVA
"MOP-IM_M06_R2"	I 4.1	BOOL	// [MOP-IM.M06]: RESERVA
"MOP-IM_M06_R3"	I 4.2	BOOL	// [MOP-IM.M06]: RESERVA
"MOP-IM_M06_R4"	I 4.3	BOOL	// [MOP-IM.M06]: RESERVA
"Z1CCFRO1"	I 10.0	BOOL	// [Z1ZB.M02]: Z1 F-RO1 CONTROL
"Z1CCFRO2"	I 10.1	BOOL	// [Z1ZB.M02]: Z1 F-RO2 CONTROL
"Z1CCB24Z"	I 10.2	BOOL	// [Z1ZB.M02]: Z1 CB 24V CONTROL (1-24Z)
"Z1CCB24R"	I 10.3	BOOL	// [Z1ZB.M02]: Z1 CB 24V CONTROL (2-24R)
"Z1ZB_M02_R1"	I 10.4	BOOL	// [Z1ZB.M02]: RESERVA
"Z1BMCY1"	I 10.5	BOOL	// [Z1ZB.M02]: CYCLE START BUTTON SOP1
"Z1BMA2"	I 10.6	BOOL	// [Z1ZB.M02]: ADVANCE BUTTON
"Z1BMR2"	I 10.7	BOOL	// [Z1ZB.M02]: RETURN BUTTON
"Z1CP7b"	I 11.0	BOOL	// [Z1ZB.M03]: Z1 EV 7 bar CONTROL
"Z1CRM"	I 11.1	BOOL	// [Z1ZB.M03]: Z1 CHECK GROUND CONTROL RELAY
"Z1ZB_M03_R1"	I 11.2	BOOL	// [Z1ZB.M03]: RESERVA
"Z1ZB_M03_R2"	I 11.3	BOOL	// [Z1ZB.M03]: RESERVA
"Z1ZB_M03_R3"	I 11.4	BOOL	// [Z1ZB.M03]: RESERVA
"Z1ZB_M03_R4"	I 11.5	BOOL	// [Z1ZB.M03]: RESERVA
"Z1ZB_M03_R5"	I 11.6	BOOL	// [Z1ZB.M03]: RESERVA
"Z1ZB_M03_R6"	I 11.7	BOOL	// [Z1ZB.M03]: RESERVA
"Z1BAUI"	I 12.0	BOOL	// [Z1ZB.M06]: Z1 FACILITY EGS (MOP/LOP)
"Z1BAU1"	I 12.1	BOOL	// [Z1ZB.M06]: PARADA EMERGENCIA SOP
"Z1SSZ"	I 12.2	BOOL	// [Z1ZB.M06]: Z1 ZONE SAFETY SELECTOR
"Z1ZB_M06_R2"	I 12.3	BOOL	// [Z1ZB.M06]: RESERVA
"Z1IFRO1"	I 23.0	BOOL	// [Z1ZB.M08]: Z1 SAFETY COMMON 1 (FRO-1 - SC1)
"Z1IFRO2"	I 24.0	BOOL	// [Z1ZB.M09]: Z1 SAFETY COMMON 2 (FRO-2 - SC2)
"Z2CCFRO1"	I 30.0	BOOL	// [Z2ZB.M02]: Z2 F-RO1 CONTROL
"Z2CCFRO2"	I 30.1	BOOL	// [Z2ZB.M02]: Z2 F-RO2 CONTROL
"Z2CCB24Z"	I 30.2	BOOL	// [Z2ZB.M02]: Z2 CB 24V CONTROL (1-24Z)
"Z2CCB24R"	I 30.3	BOOL	// [Z2ZB.M02]: Z2 CB 24V CONTROL (2-24R)
"Z2ZB_M02_R1"	I 30.4	BOOL	// [Z2ZB.M02]: RESERVA
"Z2BMCY"	I 30.5	BOOL	// [Z2ZB.M02]: Z2 START CYCLE BUTTON
"Z2BMA1"	I 30.6	BOOL	// [Z2ZB.M02]: Z2 ADVANCE BUTTON
"Z2BMR1"	I 30.7	BOOL	// [Z2ZB.M02]: Z2 RETURN BUTTON
"Z2ZB_M03_R1"	I 31.2	BOOL	// [Z2ZB.M03]: RESERVA
"Z2ZB_M03_R2"	I 31.3	BOOL	// [Z2ZB.M03]: RESERVA
"Z2ZB_M03_R3"	I 31.4	BOOL	// [Z2ZB.M03]: RESERVA
"Z2ZB_M03_R4"	I 31.5	BOOL	// [Z2ZB.M03]: RESERVA
"Z2ZB_M03_R5"	I 31.6	BOOL	// [Z2ZB.M03]: RESERVA
"Z2ZB_M03_R6"	I 31.7	BOOL	// [Z2ZB.M03]: RESERVA
"Z3CCSC1"	I 32.0	BOOL	// (Z2ZB.M02): CONTROLE RETOUR COMMUN SECUR
"Z3CCES"	I 32.1	BOOL	// (Z2ZB.M02): CONTROLE RETOUR COMMUN SECUR
"Z3CCZF"	I 32.2	BOOL	// (Z2ZB.M02): CONTROLE RETOUR COMMUN SECUR
"Z3ZB_M06_R1"	I 32.3	BOOL	// [Z2ZB.M06]: RESERVA
"Z3CCB24Z"	I 32.4	BOOL	// (Z2ZB.M02): RETOUR CONTROLE DISJONCTEUR
"Z3CCB24R"	I 32.5	BOOL	// (Z2ZB.M02): RETOUR CONTROLE DISJONCTEUR
"Z2CCB24SC"	I 32.6	BOOL	// (Z2ZB.M02): RETOUR CONTROLE DISJONCTEUR
"Z3CP7B"	I 33.0	BOOL	// (Z2ZB.M03): CONTROLE PRESSION 7 BARS
"Z3CRM"	I 33.1	BOOL	// (Z2ZB.M03): RETOUR RELAIS CONTROLE DE MA
"Z2CCB400_1"	I 33.2	BOOL	// (Z2ZB.M03): BREAKER CONTROL 400V (FROM S
"Z3BMCY"	I 34.0	BOOL	// (Z2ZB.M04): BOUTON MARCHE CYCLE
"Z3BMA1"	I 34.1	BOOL	// (Z2ZB.M04): BOUTON AVANCE MOUVEMENT
"Z3BMR1"	I 34.2	BOOL	// (Z2ZB.M04): BOUTON RECUL MOUVEMENT
"Z3BAU1"	I 35.1	BOOL	// (Z2ZB.M07): ARRET D'URGENCE ZONE
"Z3SSZ"	I 35.2	BOOL	// (Z2ZB.M07): SELECTEUR SECURITE ZONE
"ZBAUL12"	I 35.4	BOOL	// Z3B[M06] EGS Facility(LOP) 2
"Z2IFRO1"	I 43.0	BOOL	// [Z2ZB.M08]: Z2 SAFETY COMMON 1 (FRO-1 - SC1)
"Z2IFRO2"	I 44.0	BOOL	// [Z2ZB.M09]: Z2 SAFETY COMMON 2 (FRO-2 - SC2)
"A0CCFRO1"	I 70.0	BOOL	// [A0SB.M02]: A0 F-RO1 CONTROL
"A0CCFRO2"	I 70.1	BOOL	// [A0SB.M02]: A0 F-RO2 CONTROL
"A0CCFRO3"	I 70.2	BOOL	// [A0SB.M02]: A0 F-RO3 CONTROL
"A0SB_M02_R1"	I 70.3	BOOL	// [A0SB.M02]: RESERVA
"A0CCB24Z"	I 70.4	BOOL	// [A0SB.M02]: A0 CB 24V CONTROL (1-24Z)
"A0CCB24R"	I 70.5	BOOL	// [A0SB.M02]: A0 CB 24V CONTROL (2-24R)
"A0SB_M02_R2"	I 70.6	BOOL	// [A0SB.M02]: RESERVA
"A0SB_M02_R3"	I 70.7	BOOL	// [A0SB.M02]: RESERVA
"A0SB_M03_R1"	I 71.0	BOOL	// [A0SB.M03]: RESERVA
"A0SB_M03_R2"	I 71.1	BOOL	// [A0SB.M03]: RESERVA
"A0SB_M03_R3"	I 71.2	BOOL	// [A0SB.M03]: RESERVA
"A0SB_M03_R4"	I 71.3	BOOL	// [A0SB.M03]: RESERVA
"A0SB_M03_R5"	I 71.4	BOOL	// [A0SB.M03]: RESERVA
"A0SB_M03_R6"	I 71.5	BOOL	// [A0SB.M03]: RESERVA
"A0SB_M03_R7"	I 71.6	BOOL	// [A0SB.M03]: RESERVA
"A0SB_M03_R8"	I 71.7	BOOL	// [A0SB.M03]: RESERVA
"A1BAU"	I 72.0	BOOL	// [A0SB.M08]: A1 OPERATOR 1 EGS
"A2BAU"	I 72.1	BOOL	// [A0SB.M08]: A2 OPERATOR 2 EGS
"A3BAU"	I 72.2	BOOL	// [A0SB.M08]: A3 OPERATOR 3 EGS
"A0SB_M08_R1"	I 72.3	BOOL	// [A0SB.M08]: RESERVA
"A1BP1"	I 78.0	BOOL	// [A0SB.M09]: A1 T-STAND 1 BUTTON 1 (OP1) - CH1
"A1BP2"	I 78.1	BOOL	// [A0SB.M09]: A1 T-STAND 1 BUTTON 2 (OP1) - CH1
"A2BP1"	I 78.2	BOOL	// [A0SB.M09]: A2 T-STAND 2 BUTTON 1 (OP2) - CH1
"A2BP2"	I 78.3	BOOL	// [A0SB.M09]: A2 T-STAND 2 BUTTON 2 (OP2) - CH1
"A1BP12"	I 78.4	BOOL	// [A0SB.M09]: A1 T-STAND 1 BUTTON 1 (OP1) - CH2
"A1BP22"	I 78.5	BOOL	// [A0SB.M09]: A1 T-STAND 1 BUTTON 2 (OP1) - CH2
"A2BP12"	I 78.6	BOOL	// [A0SB.M09]: A2 T-STAND 2 BUTTON 1 (OP2) - CH2
"A2BP22"	I 78.7	BOOL	// [A0SB.M09]: A2 T-STAND 2 BUTTON 2 (OP2) - CH2
"A3BP1"	I 84.0	BOOL	// [A0SB.M10]: A3 T-STAND 3 BUTTON 1 (OP3) - CH1
"A3BP2"	I 84.1	BOOL	// [A0SB.M10]: A3 T-STAND 3 BUTTON 2 (OP3) - CH1
"A0SB_M10_R1"	I 84.2	BOOL	// [A0SB.M10]: RESERVA
"A0SB_M10_R2"	I 84.3	BOOL	// [A0SB.M10]: RESERVA
"A3BP12"	I 84.4	BOOL	// [A0SB.M10]: A3 T-STAND 3 BUTTON 1 (OP3) - CH2
"A3BP22"	I 84.5	BOOL	// [A0SB.M10]: A3 T-STAND 3 BUTTON 2 (OP3) - CH2
"A0SB_M10_R3"	I 84.6	BOOL	// [A0SB.M10]: RESERVA
"A0SB_M10_R4"	I 84.7	BOOL	// [A0SB.M10]: RESERVA
"A0IFRO1"	I 95.0	BOOL	// [A0SB.M12]: A0 SAFETY COMMON 1 (FRO1 - SC3)
"A0IFRO2"	I 96.0	BOOL	// [A0SB.M13]: A0 SAFETY COMMON 2 (FRO2 - SC4)
"A0IFRO3"	I 97.0	BOOL	// [A0SB.M14]: A0 SAFETY COMMON 3 (FRO3 - SC5)
"B0SB_M02_R1"	I 110.3	BOOL	// [B0SB.M02]: RESERVA
"B0SB_M02_R2"	I 110.6	BOOL	// [B0SB.M02]: RESERVA
"B0SB_M02_R3"	I 110.7	BOOL	// [B0SB.M02]: RESERVA
"B0SB_M03_R1"	I 111.0	BOOL	// [B0SB.M03]: RESERVA
"B0SB_M03_R2"	I 111.1	BOOL	// [B0SB.M03]: RESERVA
"B0SB_M03_R3"	I 111.2	BOOL	// [B0SB.M03]: RESERVA
"B0SB_M03_R4"	I 111.3	BOOL	// [B0SB.M03]: RESERVA
"B0SB_M03_R5"	I 111.4	BOOL	// [B0SB.M03]: RESERVA
"B0SB_M03_R6"	I 111.5	BOOL	// [B0SB.M03]: RESERVA
"B0SB_M03_R7"	I 111.6	BOOL	// [B0SB.M03]: RESERVA
"B0SB_M03_R8"	I 111.7	BOOL	// [B0SB.M03]: RESERVA
"B2BAU"	I 112.1	BOOL	// [B0SB.M08]: B2 OPERATOR 2 EGS
"B3BAU"	I 112.2	BOOL	// [B0SB.M08]: B3 OPERATOR 3 EGS
"B0SB_M08_R1"	I 112.3	BOOL	// [B0SB.M08]: RESERVA
"B2BP1"	I 118.2	BOOL	// [B0SB.M09]: B2 T-STAND 2 BUTTON 1 (OP2) - CH1
"B2BP2"	I 118.3	BOOL	// [B0SB.M09]: B2 T-STAND 2 BUTTON 2 (OP2) - CH1
"B2BP12"	I 118.6	BOOL	// [B0SB.M09]: B2 T-STAND 2 BUTTON 1 (OP2) - CH2
"B2BP22"	I 118.7	BOOL	// [B0SB.M09]: B2 T-STAND 2 BUTTON 2 (OP2) - CH2
"B3BP1"	I 124.0	BOOL	// [B0SB.M10]: B3 T-STAND 3 BUTTON 1 (OP3) - CH1
"B3BP2"	I 124.1	BOOL	// [B0SB.M10]: B3 T-STAND 3 BUTTON 2 (OP3) - CH1
"B0SB_M10_R1"	I 124.2	BOOL	// [B0SB.M10]: RESERVA
"B0SB_M10_R2"	I 124.3	BOOL	// [B0SB.M10]: RESERVA
"B3BP12"	I 124.4	BOOL	// [B0SB.M10]: B3 T-STAND 3 BUTTON 1 (OP3) - CH2
"B3BP22"	I 124.5	BOOL	// [B0SB.M10]: B3 T-STAND 3 BUTTON 2 (OP3) - CH2
"B0SB_M10_R3"	I 124.6	BOOL	// [B0SB.M10]: RESERVA
"B0SB_M10_R4"	I 124.7	BOOL	// [B0SB.M10]: RESERVA
"C0SB_M02_R1"	I 150.3	BOOL	// [C0SB.M02]:RESERVA
"C0SB_M02_R2"	I 150.6	BOOL	// [C0SB.M02]:RESERVA
"C0SB_M02_R3"	I 150.7	BOOL	// [C0SB.M02]:RESERVA
"C1VAL"	I 151.0	BOOL	// [C0SB.M03]: C1 OPERATOR 1 VALIDATION
"C2VAL"	I 151.1	BOOL	// [C0SB.M03]:C2 OPERATOR 2 VALIDATION
"C0SB_M03_R3"	I 151.2	BOOL	// [C0SB.M03]:RESERVA
"C0SB_M03_R4"	I 151.3	BOOL	// [C0SB.M03]:RESERVA
"C0SB_M3_R1"	I 151.4	BOOL	// [C0SB.M03]: RESERVA
"C0SB_M03_R6"	I 151.5	BOOL	// [C0SB.M03]:RESERVA
"C0SB_M03_R7"	I 151.6	BOOL	// [C0SB.M03]:RESERVA
"C0SB_M03_R8"	I 151.7	BOOL	// [C0SB.M03]:RESERVA
"C0SB_M08_R1"	I 152.2	BOOL	// [C0SB.M08]: RESERVA
"C0SB_M08_R2"	I 152.3	BOOL	// [C0SB.M08]: RESERVA
"C0SB_M09_R1"	I 158.0	BOOL	// [C0SB.M09]: RESERVA
"C0SB_M09_R2"	I 158.1	BOOL	// [C0SB.M09]: RESERVA
"C0SB_M09_R3"	I 158.2	BOOL	// [C0SB.M09]: RESERVA
"C0SB_M09_R4"	I 158.3	BOOL	// [C0SB.M09]: RESERVA
"C0SB_M09_R5"	I 158.4	BOOL	// [C0SB.M09]: RESERVA
"C0SB_M09_R6"	I 158.5	BOOL	// [C0SB.M09]: RESERVA
"C0SB_M09_R7"	I 158.6	BOOL	// [C0SB.M09]: RESERVA
"C0SB_M09_R8"	I 158.7	BOOL	// [C0SB.M09]: RESERVA
"C0SB_M10_R1"	I 164.0	BOOL	// [C0SB.M10]: RESERVA
"C0SB_M10_R2"	I 164.1	BOOL	// [C0SB.M10]: RESERVA
"C0SB_M10_R3"	I 164.2	BOOL	// [C0SB.M10]: RESERVA
"C0SB_M10_R4"	I 164.3	BOOL	// [C0SB.M10]: RESERVA
"D0CCFRO1"	I 190.0	BOOL	// [D0SB.M02]: D0 F-RO1 CONTROL
"D0CCFRO2"	I 190.1	BOOL	// [D0SB.M02]: D0 F-RO2 CONTROL
"D0CCFRO3"	I 190.2	BOOL	// [D0SB.M02]: D0 F-RO3 CONTROL
"D0SB_M02_R1"	I 190.3	BOOL	// [D0SB.M02]: RESERVA
"D0CCB24Z"	I 190.4	BOOL	// [D0SB.M02]: D0 CB 24V CONTROL (1-24Z)
"D0CCB24R"	I 190.5	BOOL	// [D0SB.M02]: D0 CB 24V CONTROL (2-24R)
"D0SB_M02_R2"	I 190.6	BOOL	// [D0SB.M02]: RESERVA
"D0SB_M02_R3"	I 190.7	BOOL	// [D0SB.M02]: RESERVA
"D0SB_M03_R1"	I 191.0	BOOL	// [D0SB.M03]: RESERVA
"D0SB_M03_R2"	I 191.1	BOOL	// [D0SB.M03]: RESERVA
"D0SB_M03_R3"	I 191.2	BOOL	// [D0SB.M03]: RESERVA
"BVLANC"	I 191.3	BOOL	// [D0SB.M03]: BOTON VALIDACIÓN LANZAMIENTO
"D0SB_M03_R5"	I 191.4	BOOL	// [D0SB.M03]: RESERVA
"D0SB_M03_R6"	I 191.5	BOOL	// [D0SB.M03]: RESERVA
"D0SB_M03_R7"	I 191.6	BOOL	// [D0SB.M03]: RESERVA
"D0SB_M03_R8"	I 191.7	BOOL	// [D0SB.M03]: RESERVA
"D1BAU"	I 192.0	BOOL	// [D0SB.M08]: D1 OPERATOR 1 EGS
"D2BAU"	I 192.1	BOOL	// [D0SB.M08]: D2 OPERATOR 2 EGS
"D3BAU"	I 192.2	BOOL	// [D0SB.M08]: D3 OPERATOR 3 EGS
"D4BAU"	I 192.3	BOOL	// [D0SB.M08]: D4 OPERATOR 4 EGS
"D1BP1"	I 198.0	BOOL	// [D0SB.M09]: D1 T-STAND 1 BUTTON 1 (OP1) - CH1
"D1BP2"	I 198.1	BOOL	// [D0SB.M09]: D1 T-STAND 1 BUTTON 2 (OP1) - CH1
"D2BP1"	I 198.2	BOOL	// [D0SB.M09]: D2 T-STAND 2 BUTTON 1 (OP2) - CH1
"D2BP2"	I 198.3	BOOL	// [D0SB.M09]: D2 T-STAND 2 BUTTON 2 (OP2) - CH1
"D1BP12"	I 198.4	BOOL	// [D0SB.M09]: D1 T-STAND 1 BUTTON 1 (OP1) - CH2
"D1BP22"	I 198.5	BOOL	// [D0SB.M09]: D1 T-STAND 1 BUTTON 2 (OP1) - CH2
"D2BP12"	I 198.6	BOOL	// [D0SB.M09]: D2 T-STAND 2 BUTTON 1 (OP2) - CH2
"D2BP22"	I 198.7	BOOL	// [D0SB.M09]: D2 T-STAND 2 BUTTON 2 (OP2) - CH2
"D3BP1"	I 204.0	BOOL	// [D0SB.M10]: D3 T-STAND 3 BUTTON 1 (OP3) - CH1
"D3BP2"	I 204.1	BOOL	// [D0SB.M10]: D3 T-STAND 3 BUTTON 2 (OP3) - CH1
"D4BP1"	I 204.2	BOOL	// [D0SB.M10]: D4 T-STAND 4 BUTTON 1 (OP4) - CH1
"D4BP2"	I 204.3	BOOL	// [D0SB.M10]: D4 T-STAND 4 BUTTON 2 (OP4) - CH1
"D3BP12"	I 204.4	BOOL	// [D0SB.M10]: D3 T-STAND 3 BUTTON 1 (OP3) - CH2
"D3BP22"	I 204.5	BOOL	// [D0SB.M10]: D3 T-STAND 3 BUTTON 2 (OP3) - CH2
"D4BP12"	I 204.6	BOOL	// [D0SB.M10]: D4 T-STAND 4 BUTTON 1 (OP4) - CH2
"D4BP22"	I 204.7	BOOL	// [D0SB.M10]: D4 T-STAND 4 BUTTON 2 (OP4) - CH2
"D0IFRO1"	I 215.0	BOOL	// [D0SB.M12]: D0 SAFETY COMMON 1 (FRO-1 - SC3)
"D0IFRO2"	I 216.0	BOOL	// [D0SB.M13]: D0 SAFETY COMMON 2 (FRO-2 - SC4)
"D0IFRO3"	I 217.0	BOOL	// [D0SB.M14]: D0 SAFETY COMMON 3 (FRO-3 - SC5)
"F0CCFRO1"	I 270.0	BOOL	// [F0SB.M02]: F0 F-RO1 CONTROL
"F0CCFRO2"	I 270.1	BOOL	// [F0SB.M02]: F0 F-RO2 CONTROL
"F0CCFRO3"	I 270.2	BOOL	// [F0SB.M02]: F0 F-RO3 CONTROL
"F0SB_M02_R1"	I 270.3	BOOL	// [F0SB.M02]: RESERVA
"F0CCB24Z"	I 270.4	BOOL	// [F0SB.M02]: F0 CB 24V CONTROL (1-24Z)
"F0CCB24R"	I 270.5	BOOL	// [F0SB.M02]: F0 CB 24V CONTROL (2-24R)
"F0SB_M02_R2"	I 270.6	BOOL	// [F0SB.M02]: RESERVA
"F0SB_M02_R3"	I 270.7	BOOL	// [F0SB.M02]: RESERVA
"F0SB_M03_R1"	I 271.0	BOOL	// [F0SB.M03]: RESERVA
"F0SB_M03_R2"	I 271.1	BOOL	// [F0SB.M03]: RESERVA
"F0SB_M03_R3"	I 271.2	BOOL	// [F0SB.M03]: RESERVA
"F0SB_M03_R4"	I 271.3	BOOL	// [F0SB.M03]: RESERVA
"F0SB_M03_R5"	I 271.4	BOOL	// [F0SB.M03]: RESERVA
"F0SB_M03_R6"	I 271.5	BOOL	// [F0SB.M03]: RESERVA
"F0SB_M03_R7"	I 271.6	BOOL	// [F0SB.M03]: RESERVA
"F0SB_M03_R8"	I 271.7	BOOL	// [F0SB.M03]: RESERVA
"F1BAU"	I 272.0	BOOL	// [F0SB.M08]: F1 OPERATOR 1 EGS
"F2BAU"	I 272.1	BOOL	// [F0SB.M08]: F2 OPERATOR 2 EGS
"F3BAU"	I 272.2	BOOL	// [F0SB.M08]: F3 OPERATOR 3 EGS
"F0SB_M08_R1"	I 272.3	BOOL	// [F0SB.M08]: RESERVA
"F1BP1"	I 278.0	BOOL	// [F0SB.M09]: F1 T-STAND 1 BUTTON 1 (OP1) - CH1
"F1BP2"	I 278.1	BOOL	// [F0SB.M09]: F1 T-STAND 1 BUTTON 2 (OP1) - CH1
"F2BP1"	I 278.2	BOOL	// [F0SB.M09]: F2 T-STAND 2 BUTTON 1 (OP2) - CH1
"F2BP2"	I 278.3	BOOL	// [F0SB.M09]: F2 T-STAND 2 BUTTON 2 (OP2) - CH1
"F1BP12"	I 278.4	BOOL	// [F0SB.M09]: F1 T-STAND 1 BUTTON 1 (OP1) - CH2
"F1BP22"	I 278.5	BOOL	// [F0SB.M09]: F1 T-STAND 1 BUTTON 2 (OP1) - CH2
"F2BP12"	I 278.6	BOOL	// [F0SB.M09]: F2 T-STAND 2 BUTTON 1 (OP2) - CH2
"F2BP22"	I 278.7	BOOL	// [F0SB.M09]: F2 T-STAND 2 BUTTON 2 (OP2) - CH2
"F3BP1"	I 284.0	BOOL	// [F0SB.M10]: F3 T-STAND 3 BUTTON 1 (OP3) - CH1
"F3BP2"	I 284.1	BOOL	// [F0SB.M10]: F3 T-STAND 3 BUTTON 2 (OP3) - CH1
"F0SB_M10_R1"	I 284.2	BOOL	// [F0SB.M10]: RESERVA
"F0SB_M10_R2"	I 284.3	BOOL	// [F0SB.M10]: RESERVA
"F3BP12"	I 284.4	BOOL	// [F0SB.M10]: F3 T-STAND 3 BUTTON 1 (OP3) - CH2
"F3BP22"	I 284.5	BOOL	// [F0SB.M10]: F3 T-STAND 3 BUTTON 2 (OP3) - CH2
"F0SB_M10_R3"	I 284.6	BOOL	// [F0SB.M10]: RESERVA
"F0SB_M10_R4"	I 284.7	BOOL	// [F0SB.M10]: RESERVA
"F0IFRO1"	I 295.0	BOOL	// [F0SB.M12]: F0 SAFETY COMMON 1 (FRO-1 - SC3)
"F0IFRO2"	I 296.0	BOOL	// [F0SB.M13]: F0 SAFETY COMMON 2 (FRO-2 - SC4)
"F0IFRO3"	I 297.0	BOOL	// [F0SB.M14]: F0 SAFETY COMMON 3 (FRO-3 - SC5)
"RES3"	I 351.3	BOOL	// [H0SB.M03]: RESERVA
"H1BAU"	I 352.0	BOOL	// [H0SB.M08]: H1 OPERATOR 1 EGS
"H2BAU"	I 352.1	BOOL	// [H0SB.M08]: H2 OPERATOR 2 EGS
"H1BP1"	I 358.0	BOOL	// [H0SB.M09]: H1 T-STAND 1 BUTTON 1 (OP1) - CH1
"H1BP2"	I 358.1	BOOL	// [H0SB.M09]: H1 T-STAND 1 BUTTON 2 (OP1) - CH1
"H2BP1"	I 358.2	BOOL	// [H0SB.M09]: H2 T-STAND 2 BUTTON 1 (OP2) - CH1
"H2BP2"	I 358.3	BOOL	// [H0SB.M09]: H2 T-STAND 2 BUTTON 2 (OP2) - CH1
"H1BP12"	I 358.4	BOOL	// [H0SB.M09]: H1 T-STAND 1 BUTTON 1 (OP1) - CH2
"H1BP22"	I 358.5	BOOL	// [H0SB.M09]: H1 T-STAND 1 BUTTON 2 (OP1) - CH2
"H2BP12"	I 358.6	BOOL	// [H0SB.M09]: H2 T-STAND 2 BUTTON 1 (OP2) - CH2
"H2BP22"	I 358.7	BOOL	// [H0SB.M09]: H2 T-STAND 2 BUTTON 2 (OP2) - CH2
"K0CCFRO1"	I 378.0	BOOL	// [K0SB.M02]: K0 F-RO1 CONTROL
"K0CCFRO2"	I 378.1	BOOL	// [K0SB.M02]: K0 F-RO2 CONTROL
"K0CCFRO3"	I 378.2	BOOL	// [K0SB.M02]: K0 F-RO3 CONTROL
"K0SB_M02_R1"	I 378.3	BOOL	// [K0SB.M02]: RESERVA
"K0CCB24Z"	I 378.4	BOOL	// [K0SB.M02]: K0 CB 24V CONTROL (2-24Z)
"K0CCB24R"	I 378.5	BOOL	// [K0SB.M02]: K0 CB 24V CONTROL (2-24R)
"K0SB_M02_R2"	I 378.6	BOOL	// [K0SB.M02]: RESERVA
"K0SB_M02_R3"	I 378.7	BOOL	// [K0SB.M02]: RESERVA
"K0SB_M03_R1"	I 379.0	BOOL	// [K0SB.M03]: RESERVA
"K0SB_M03_R2"	I 379.1	BOOL	// [K0SB.M03]: RESERVA
"K0SB_M03_R3"	I 379.2	BOOL	// [K0SB.M03]: RESERVA
"K0SB_M03_R4"	I 379.3	BOOL	// [K0SB.M03]: RESERVA
"K0SB_M03_R5"	I 379.4	BOOL	// [K0SB.M03]: RESERVA
"K0SB_M03_R6"	I 379.5	BOOL	// [K0SB.M03]: RESERVA
"K0SB_M03_R7"	I 379.6	BOOL	// [K0SB.M03]: RESERVA
"K0SB_M03_R8"	I 379.7	BOOL	// [K0SB.M03]: RESERVA
"K1BAU"	I 382.0	BOOL	// [K0SB.M08]: K1 OPERATOR 1 EGS
"K2BAU"	I 382.1	BOOL	// [K0SB.M08]: K1 OPERATOR 2 EGS
"K0SB_M08_R1"	I 382.2	BOOL	// [K0SB.M08]: RESERVA
"K0SB_M08_R2"	I 382.3	BOOL	// [K0SB.M08]: RESERVA
"K1BP1"	I 388.0	BOOL	// [K0SB.M09]: K1 T-STAND 1 BUTTON 1 (OP1) - CH1
"K1BP2"	I 388.1	BOOL	// [K0SB.M09]: K1 T-STAND 1 BUTTON 2 (OP1) - CH1
"K0SB_M09_R3"	I 388.2	BOOL	// [K0SB.M09]: RESERVA
"K0SB_M09_R4"	I 388.3	BOOL	// [K0SB.M09]: RESERVA
"K1BP12"	I 388.4	BOOL	// [K0SB.M09]: K1 T-STAND 1 BUTTON 1 (OP1) - CH2
"K1BP22"	I 388.5	BOOL	// [K0SB.M09]: K1 T-STAND 1 BUTTON 2 (OP1) - CH2
"K0SB_M09_R7"	I 388.6	BOOL	// [K0SB.M09]: RESERVA
"K0SB_M09_R8"	I 388.7	BOOL	// [K0SB.M09]: RESERVA
"K0SB_M10_R1"	I 394.0	BOOL	// [K0SB.M10]: RESERVA
"K0SB_M10_R2"	I 394.1	BOOL	// [K0SB.M10]: RESERVA
"K0SB_M10_R3"	I 394.2	BOOL	// [K0SB.M10]: RESERVA
"K0SB_M10_R4"	I 394.3	BOOL	// [K0SB.M10]: RESERVA
"K0IFRO1"	I 405.0	BOOL	// [K0SB.M12]: K0 SAFETY COMMON 1 (FRO1 - SC3)
"K0IFRO2"	I 406.0	BOOL	// [K0SB.M13]: K0 SAFETY COMMON 2 (FRO2 - SC4)
"K0IFRO3"	I 407.0	BOOL	//  [K0SB.M14]: K0 SAFETY COMMON 3 (FRO3 - SC5)
"A0DPP1"	I 500.0	BOOL	// [A0IM1.A0E11]: A0: DETECTOR PRESENÇA DE PEÇA 1
"A0DPP3"	I 500.1	BOOL	// [A0IM1.A0E11]: A0: DETECTOR PRESENÇA DE PEÇA 3
"A0DPP5"	I 500.2	BOOL	// [A0IM1.A0E11]: A0: DETECTOR PRESENÇA DE PEÇA 5
"A0DPP7"	I 500.3	BOOL	// [A0IM1.A0E11]: A0: DETECTOR PRESENÇA DE PEÇA 7
"A0DPP2"	I 500.4	BOOL	// [A0IM1.A0E11]: A0: DETECTOR PRESENÇA DE PEÇA 2
"A0DPP4"	I 500.5	BOOL	// [A0IM1.A0E11]: A0: DETECTOR PRESENÇA DE PEÇA 4
"A0DPP6"	I 500.6	BOOL	// [A0IM1.A0E11]: A0: DETECTOR PRESENÇA DE PEÇA 6
"A0DPP8"	I 500.7	BOOL	// [A0IM1.A0E11]: A0: DETECTOR PRESENÇA DE PEÇA 8
"A0DPP9"	I 501.0	BOOL	// [A0IM1.A0E12]: A0: DETECTOR PRESENÇA DE PEÇA 9
"A0IM_A0E12_R1"	I 501.1	BOOL	// [A0IM1.A0E12]: RESERVA
"A0DAPLA1"	I 501.2	BOOL	// [A0IM1.A0E12]: A0:DETECTOR AVANC0 PILOTO A1
"A0DAPLA2"	I 501.3	BOOL	// [A0IM1.A0E12]: A0:DETECTOR AVANCO PILOTO A2
"A0DPP10"	I 501.4	BOOL	// [A0IM1.A0E12]: A0: DETECTOR PRESENÇA DE PEÇA 10
"A0IM_A0E12_R2"	I 501.5	BOOL	// [A0IM1.A0E12]: RESERVA
"A0DRPLA1"	I 501.6	BOOL	// [A0IM1.A0E12]: A0:DETECTOR RECUO PILOTO A1
"A0DRPLA2"	I 501.7	BOOL	// [A0IM1.A0E12]: A0:DETECTOR RECUO PILOTO A2
"A0DRPLE1"	I 502.0	BOOL	// [A0IM1.A0E13]: A0:DETECTOR RECUO PILOTO E1
"A0DRPLE2"	I 502.1	BOOL	// [A0IM1.A0E13]: A0:DETECTOR RECUO PILOTO E2
"A0DRSRB1"	I 502.2	BOOL	// [A0IM1.A0E13]: A0: DETECTOR RECUO SERRAGE MANUAL B1
"A0DRSRB2"	I 502.3	BOOL	// [A0IM1.A0E13]: A0: DETECTOR  RECUO SERRAGE MANUAL B2
"A0DAPLE1"	I 502.4	BOOL	// [A0IM1.A0E13]: A0:DETECTOR AVANÇO PILOTO E1
"A0DAPLE2"	I 502.5	BOOL	// [A0IM1.A0E13]: A0:DETECTOR AVANÇO PILOTO E2
"A0DASRB1"	I 502.6	BOOL	// [A0IM1.A0E13]: A0: DETECTOR AVANÇO SERRAGE MANUAL B1
"A0DASRB2"	I 502.7	BOOL	// [A0IM1.A0E13]: A0: DETECTOR AVANÇO SERRAGE MANUAL B2
"A0DRSRD1"	I 503.0	BOOL	// [A0IM1.A0E14]: A0: DETECTOR RECUO SERRAGE D1
"A0DRSRD2"	I 503.1	BOOL	// [A0IM1.A0E14]: A0: DETECTOR RECUO SERRAGE D2
"A0DRSRD3"	I 503.2	BOOL	// [A0IM1.A0E14]: A0: DETECTOR RECUO SERRAGE D3
"A0DRSRD4"	I 503.3	BOOL	// [A0IM1.A0E14]: A0: DETECTOR RECUO SERRAGE D4
"A0DASRD1"	I 503.4	BOOL	// [A0IM1.A0E14]: A0: DETECTOR AVANÇO SERRAGE D1
"A0DASRD2"	I 503.5	BOOL	// [A0IM1.A0E14]: A0: DETECTOR AVANÇO SERRAGE D2
"A0DASRD3"	I 503.6	BOOL	// [A0IM1.A0E14]: A0: DETECTOR AVANÇO SERRAGE D3
"A0DASRD4"	I 503.7	BOOL	// [A0IM1.A0E14]: A0: DETECTOR AVANÇO SERRAGE D4
"A0DCZA"	I 504.0	BOOL	// A0: Detector Guinche Zona A (Cruzeta)
"A0IM_A0E15_R2"	I 504.1	BOOL	// [A0IM1.A0E15]: RESERVA
"A0IM_A0E15_R3"	I 504.2	BOOL	// [A0IM1.A0E15]: RESERVA
"A0IM_A0E15_R4"	I 504.3	BOOL	// [A0IM1.A0E15]: RESERVA
"A0IM_A0E15_R5"	I 504.4	BOOL	// [A0IM1.A0E15]: RESERVA
"A0IM_A0E15_R6"	I 504.5	BOOL	// [A0IM1.A0E15]: RESERVA
"A0IM_A0E15_R7"	I 504.6	BOOL	// [A0IM1.A0E15]: RESERVA
"A0IM_A0E15_R8"	I 504.7	BOOL	// [A0IM1.A0E15]: RESERVA
"B0IM_B0E11_R1"	I 520.1	BOOL	// [B0IM1.B0E11]: RESERVA
"B0DAPLA1"	I 520.2	BOOL	// [B0IM1.B0E11]: B0:DETECTOR RECUO PILOTO A1
"B0DAPLA2"	I 520.3	BOOL	// [B0IM1.B0E11]: B0:DETECTOR RECUO PILOTO A2
"B0IM_B0E11_R2"	I 520.4	BOOL	// [B0IM1.B0E11]: RESERVA
"B0IM_B0E11_R3"	I 520.5	BOOL	// [B0IM1.B0E11]: RESERVA
"B0DRPLA1"	I 520.6	BOOL	// [B0IM1.B0E11]: B0:DETECTOR AVANÇO PILOTO A1
"B0DRPLA2"	I 520.7	BOOL	// [B0IM1.B0E11]: B0:DETECTOR AVANÇO PILOTO A2
"B0DRSRB1"	I 521.0	BOOL	// [B0IM1.B0E12]: B0: DETECTOR RECUO SERRAGE B1
"B0DRSRB2"	I 521.1	BOOL	// [B0IM1.B0E12]: B0: DETECTOR RECUO SERRAGE B2
"B0IM_B0E12_R1"	I 521.2	BOOL	// [B0IM1.B0E12]: RESERVA
"B0IM_B0E12_R2"	I 521.3	BOOL	// [B0IM1.B0E12]: RESERVA
"B0DASRB1"	I 521.4	BOOL	// [B0IM1.B0E12]: B0: DETECTOR AVANÇO SERRAGE B1
"B0DASRB2"	I 521.5	BOOL	// [B0IM1.B0E12]: B0: DETECTOR AVANÇO SERRAGE B2
"B0IM_B0E12_R3"	I 521.6	BOOL	// [B0IM1.B0E12]: RESERVA
"B0IM_B0E12_R4"	I 521.7	BOOL	// [B0IM1.B0E12]: RESERVA
"C0IM_C0E11_R1"	I 540.1	BOOL	// [C0IM1.C0E11]: RESERVA
"C0IM_C0E11_R2"	I 540.2	BOOL	// [C0IM1.C0E11]: RESERVA
"C0IM_C0E11_R3"	I 540.3	BOOL	// [C0IM1.C0E11]: RESERVA
"C0IM_C0E11_R4"	I 540.4	BOOL	// [C0IM1.C0E11]: RESERVA
"C0IM_C0E11_R5"	I 540.5	BOOL	// [C0IM1.C0E11]: RESERVA
"C0IM_C0E11_R6"	I 540.6	BOOL	// [C0IM1.C0E11]: RESERVA
"C0IM_C0E11_R7"	I 540.7	BOOL	// [C0IM1.C0E11]: RESERVA
"D0DPP1"	I 560.0	BOOL	// [D0IM1.D0E11]: D0: DETECTOR PRESENÇA DE PEÇA 1
"D0DPP3"	I 560.1	BOOL
"D0DPP5"	I 560.2	BOOL	// [D0IM1.D0E11]: D0: DETECTOR PRESENÇA DE PEÇA 5
"D0DPP7"	I 560.3	BOOL	// [D0IM1.D0E11]: D0: DETECTOR PRESENÇA DE PEÇA 7
"D0DPP2"	I 560.4	BOOL	// [D0IM1.D0E11]: D0: DETECTOR PRESENÇA DE PEÇA 2
"D0DPP4"	I 560.5	BOOL	// [D0IM1.D0E11]: D0: DETECTOR PRESENÇA DE PEÇA 4
"D0DPP6"	I 560.6	BOOL	// [D0IM1.D0E11]: D0: DETECTOR PRESENÇA DE PEÇA 6
"D0DPP8"	I 560.7	BOOL	// [D0IM1.D0E11]: D0: DETECTOR PRESENÇA DE PEÇA 8
"D0DPP9"	I 561.0	BOOL	// [D0IM1.D0E12]: D0: DETECTOR PRESENÇA DE PEÇA 9
"D0IM_D0E12_R1"	I 561.1	BOOL	// [D0IM1.D0E12]: RESERVA
"D0DAPLA1"	I 561.2	BOOL	// [D0IM1.D0E12]: D0:DETECTOR AVANÇO PILOTO A1
"D0DAPLA2"	I 561.3	BOOL	// [D0IM1.D0E12]: D0:DETECTOR AVANÇO PILOTO A2
"D0IM_D0E12_R2"	I 561.4	BOOL	// [D0IM1.D0E12]: RESERA
"D0IM_D0E12_R3"	I 561.5	BOOL	// [D0IM1.D0E12]: RESERVA
"D0DRPLA1"	I 561.6	BOOL	// [D0IM1.D0E12]: D0:DETECTOR RECUO PILOTO A1
"D0DRPLA2"	I 561.7	BOOL	// [D0IM1.D0E12]: D0:DETECTOR  RECUO PILOTO A2
"D0DRPLE1"	I 562.0	BOOL	// [D0IM1.D0E13]: D0:DETECTOR RECUO PILOTO E1
"D0DRPLE2"	I 562.1	BOOL	// [D0IM1.D0E13]: D0:DETECTOR RECUO PILOTO E2
"D0DRCAB1"	I 562.2	BOOL	// [D0IM1.D0E13]: D0:DETECTOR RECUO CARRO B1
"D0DRCAB2"	I 562.3	BOOL	// [D0IM1.D0E13]: D0:DETECTOR RECUO CARRO B2
"D0DAPLE1"	I 562.4	BOOL	// [D0IM1.D0E13]: D0:DETECTOR AVANÇO PILOTO E1
"D0DAPLE2"	I 562.5	BOOL	// [D0IM1.D0E13]: D0:DETECTOR AVANÇO PILOTO E2
"D0DACAB1"	I 562.6	BOOL	// [D0IM1.D0E13]: D0:DETECTOR AVANÇO CARRO B1
"D0DACAB2"	I 562.7	BOOL	// [D0IM1.D0E13]: D0:DETECTOR AVANÇO CARRO B2
"D0DRSRC1"	I 563.0	BOOL	// [D0IM1.D0E14]: D0: DETECTOR RECUO SERRAGE C1
"D0DRSRC2"	I 563.1	BOOL	// [D0IM1.D0E14]: D0: DETECTOR RECUO SERRAGE C2
"D0DRSRC3"	I 563.2	BOOL	// [D0IM1.D0E14]: D0: DETECTOR RECUO SERRAGE C3
"D0DRSRC4"	I 563.3	BOOL	// [D0IM1.D0E14]: D0: DETECTOR RECUO SERRAGE C4
"D0DASRC1"	I 563.4	BOOL	// [D0IM1.D0E14]: D0: DETECTOR AVANÇO SERRAGE C1
"D0DASRC2"	I 563.5	BOOL	// [D0IM1.D0E14]: D0: DETECTOR AVANÇO SERRAGE C2
"D0DASRC3"	I 563.6	BOOL	// [D0IM1.D0E14]: D0: DETECTOR AVANÇO SERRAGE C3
"D0DASRC4"	I 563.7	BOOL	// [D0IM1.D0E14]: D0: DETECTOR AVANÇO SERRAGE C4
"D0DRSRD1"	I 564.0	BOOL	// [D0IM1.D0E15]: D0: DETECTOR RECUO SERRAGE D1
"D0DRSRD2"	I 564.1	BOOL	// [D0IM1.D0E15]: D0: DETECTOR RECUO SERRAGE D2
"D0DRSRD3"	I 564.2	BOOL	// [D0IM1.D0E15]: D0: DETECTOR RECUO SERRAGE D3
"D0DPP11"	I 564.3	BOOL	// [D0IM1.D0E15]: DETECTOR PRESENCIA DE PIEZA 11
"D0DASRD1"	I 564.4	BOOL	// [D0IM1.D0E15]: D0: DETECTOR AVANÇO SERRAGE D1
"D0DASRD2"	I 564.5	BOOL	// [D0IM1.D0E15]: D0: DETECTOR AVANÇO SERRAGE D2
"D0DASRD3"	I 564.6	BOOL	// [D0IM1.D0E15]: D0: DETECTOR AVANÇO SERRAGE D3
"D0DPP12"	I 564.7	BOOL	// [D0IM1.D0E15]: DETECTOR PRESENCIA DE PIEZA 12
"D0FT2DPP"	I 565.0	BOOL	// [D0IM1.D0E16]: FOTOCELULA 2 DETECTORA DE PRESENÇA DE PEÇA
"D0FT1DPP"	I 565.1	BOOL	// [D0IM1.D0E16]: FOTOCELULA 1 DETECTORA DE PRESENÇA DE PEÇA
"D0DRSRMF1"	I 565.2	BOOL	// [D0IM1.D0E16]: Detector Retroceso SRM1
"D0DCZA"	I 565.3	BOOL	// [D0IM1.D0E16]: Detector Guinche Zona A (Cruzeta)
"D0IN_D0E16_R5"	I 565.4	BOOL	// [D0IM1.D0E16]: RESERVA
"D0IN_D0E16_R6"	I 565.5	BOOL	// [D0IM1.D0E16]: RESERVA
"D0DASRMF1"	I 565.6	BOOL	// [D0IM1.D0E16]: Detector Avance SRM1
"D0DCZB"	I 565.7	BOOL	// [D0IM1.D0E16]: Detector Guinche Zona B (Cruzeta)
"E0DPP3"	I 580.1	BOOL	// [E0IM1.E0E11]: E0: DETECTOR PRESENÇA DE PEÇA 3
"E0DAPLA1"	I 580.2	BOOL	// [E0IM1.E0E11]: E0:DETECTOR AVANÇO PILOTO A1
"E0DAPLA2"	I 580.3	BOOL	// [E0IM1.E0E11]: E0:DETECTOR AVANÇO PILOTO A2
"E0DPP2"	I 580.4	BOOL	// [E0IM1.E0E11]: E0: DETECTOR PRESENÇA DE PEÇA 2
"E0IM_E0E11_R1"	I 580.5	BOOL	// [E0IM1.E0E11]: RESERVA
"E0DRPLA1"	I 580.6	BOOL	// [E0IM1.E0E11]: E0:DETECTOR RECUO PILOTO A1
"E0DRPLA2"	I 580.7	BOOL	// [E0IM1.E0E11]: E0:DETECTOR RECUO PILOTO A2
"E0DRSRB1"	I 581.0	BOOL	// [E0IM1.E0E12]: E0: DETECTOR RECUO SERRAGE B1
"E0DRSRB2"	I 581.1	BOOL	// [E0IM1.E0E12]: E0: DETECTOR RECUO SERRAGE B2
"E0IM1_E0E12_R1"	I 581.2	BOOL	// [E0IM1.E0E12]: RESERVA
"E0IM1_E0E12_R2"	I 581.3	BOOL	// [E0IM1.E0E12]: RESERVA
"E0DASRB1"	I 581.4	BOOL	// [E0IM1.E0E12]: E0: DETECTOR AVANÇO SERRAGE B1
"E0DASRB2"	I 581.5	BOOL	// [E0IM1.E0E12]: E0: DETECTOR AVANÇO SERRAGE B2
"E0IM1_E0E12_R3"	I 581.6	BOOL	// [E0IM1.E0E12]: RESERVA
"E0IM1_E0E12_R4"	I 581.7	BOOL	// [E0IM1.E0E12]: RESERVA
"F0DPP1"	I 600.0	BOOL	// [F0IM1.F0E11]: F0: DETECTOR PRESENÇA DE PEÇA 1
"F0IM_F0E11_R1"	I 600.1	BOOL	// [F0IM1.F0E11]: RESERVA
"F0DPP3"	I 600.2	BOOL	// [F0IM1.F0E11]: F0:  DETECTOR DIV B52-B52 CROSS/ L52 4
"F0DPP4"	I 600.3	BOOL	// [F0IM1.F0E11]: FO:DETECTOR PRESENCIA DE PIEZA 3
"F0DPP2"	I 600.4	BOOL	// [F0IM1.F0E11]: F0: DETECTOR PRESENÇA DE PEÇA 2
"F0IM_F0E11_R4"	I 600.5	BOOL	// [F0IM1.F0E11]: RESERVA
"F0DPP5"	I 600.6	BOOL	// [F0IM1.F0E11]: F0: DETECTOR PRESENCIA DE PIEZA 5
"F0IM_F0E11_R6"	I 600.7	BOOL	// [F0IM1.F0E11]: RESERVA
"F0DAPLA1"	I 601.0	BOOL	// [F0IM1.F0E12]: F0:DETECTOR AVANÇO PILOTO A1
"F0DAPLA2"	I 601.1	BOOL	// [F0IM1.F0E12]: F0:DETECTOR AVANÇO PILOTO A2
"F0DRPLA3"	I 601.2	BOOL	// [F0IM1.F0E12]: F0:DETECTOR RECUO PILOTO A3
"F0DRPLA4"	I 601.3	BOOL	// [F0IM1.F0E12]: F0:DETECTOR RECUO PILOTO A4
"F0DRPLA1"	I 601.4	BOOL	// [F0IM1.F0E12]: F0:DETECTOR  RECUO  PILOTO A1
"F0DRPLA2"	I 601.5	BOOL	// [F0IM1.F0E12]: F0:DETECTOR  RECUO  PILOTO A2
"F0DAPLA3"	I 601.6	BOOL	// [F0IM1.F0E12]: F0:DETECTOR AVANÇO PILOTO A3
"F0DAPLA4"	I 601.7	BOOL	// [F0IM1.F0E12]: F0:DETECTOR AVANÇO PILOTO A4
"F0DRPLA5"	I 602.0	BOOL	// [F0IM1.F0E13]: F0:DETECTOR RECUO PILOTO A5
"F0DRPLA6"	I 602.1	BOOL	// [F0IM1.F0E13]: F0:DETECTOR RECUO PILOTO A6
"F0DRSRB1"	I 602.2	BOOL	// [F0IM1.F0E13]: F0: DETECTOR RECUO SERRAGE MANUAL B1
"F0DRSRB2"	I 602.3	BOOL	// [F0IM1.F0E13]: F0: DETECTOR RECUO SERRAGE MANUAL B2
"F0DAPLA5"	I 602.4	BOOL	// [F0IM1.F0E13]: F0:DETECTOR AVANÇO PILOTO A5
"F0DAPLA6"	I 602.5	BOOL	// [F0IM1.F0E13]: F0:DETECTOR AVANÇO PILOTO A6
"F0DASRB1"	I 602.6	BOOL	// [F0IM1.F0E13]: F0: DETECTOR AVANÇO SERRAGE MANUAL B1
"F0DASRB2"	I 602.7	BOOL	// [F0IM1.F0E13]: F0: DETECTOR AVANÇO SERRAGE MANUAL B2
"F0DRSRD1"	I 603.0	BOOL	// [F0IM1.F0E14]: F0: DETECTOR RECUO SERRAGE D1
"F0DRSRD2"	I 603.1	BOOL	// [F0IM1.F0E14]: F0: DETECTOR RECUO SERRAGE D2
"F0DRRCE1"	I 603.2	BOOL	// [F0IM1.F0E14]: F0: DETECTOR RECUO RETACAGE E1
"F0DRRCE2"	I 603.3	BOOL	// [F0IM1.F0E14]: F0: DETECTOR RECUO RETACAGE E2
"F0DASRD1"	I 603.4	BOOL	// [F0IM1.F0E14]: F0: DETECTOR AVANÇO SERRAGE D1
"F0DASRD2"	I 603.5	BOOL	// [F0IM1.F0E14]: F0: DETECTOR AVANÇO SERRAGE D2
"F0DARCE1"	I 603.6	BOOL	// [F0IM1.F0E14]: F0: DETECTOR AVANÇO RETACAGE E1
"F0DARCE2"	I 603.7	BOOL	// [F0IM1.F0E14]: F0: DETECTOR AVANÇO RETACAGE E2
"F0DACAF1"	I 604.0	BOOL	// [F0IM1.F0E15]: F0: DETECTOR AVANÇO CARRO F1
"F0DICAF1"	I 604.1	BOOL	// [F0IM1.F0E15]: F0: DETECTOR INTERMEDIARIO CARRO F1
"F0IM_F0E15_R2"	I 604.2	BOOL	// [F0IM1.F0E15]: RESERVA
"F0DCZA"	I 604.3	BOOL	// [F0IM1.F0E15]: Detector Guinche Zona A (Cruzeta)
"F0DRCAF1"	I 604.4	BOOL	// [F0IM1.F0E15]: F0: DETECTOR RECUO CARRO F1
"F0IM_F0E15_R4"	I 604.5	BOOL	// [F0IM1.F0E15]: RESERVA
"F0IM_F0E15_R5"	I 604.6	BOOL	// [F0IM1.F0E15]: RESERVA
"F0DCZB"	I 604.7	BOOL	// [F0IM1.F0E15]: Detector Guinche Zona B (Cruzeta)
"G0DAPLA1"	I 620.1	BOOL	// [G0IM1.G0E11]: G0: DETECTOR AVANÇO PILOTO A1
"G0DAPLA2"	I 620.2	BOOL	// [G0IM1.G0E11]: G0: DETECTOR AVANÇO PILOTO A2
"G0DRSRB1"	I 620.3	BOOL	// [G0IM1.G0E11]: G0: DETECTOR RECUO SERRAGE B1
"G0DRPLA1"	I 620.5	BOOL	// [G0IM1.G0E11]: G0: DETECTOR RECUO PILOTO A1
"G0DRPLA2"	I 620.6	BOOL	// [G0IM1.G0E11]: G0: DETECTOR RECUO PILOTO A2
"G0DASRB1"	I 620.7	BOOL	// [G0IM1.G0E11]: G0: DETECTOR AVANÇO SERRAGE B1
"G0DRSRB2"	I 621.0	BOOL	// [G0IM1.G0E12]: G0: DETECTOR RECUO SERRAGE B2
"CT_M6_03_FAG0039"	I 621.1	BOOL	// Contagem de tucker M6 pistola 3 do DCE FAG0039
"G0IM_G0E12_R2"	I 621.2	BOOL	// [G0IM1.G0E12]: RESERVA
"G0IM_G0E12_R3"	I 621.3	BOOL	// [G0IM1.G0E12]: RESERVA
"G0DASRB2"	I 621.4	BOOL	// [G0IM1.G0E12]: G0: DETECTOR AVANÇO SERRAGE B2
"CT_M6_01_FAG0014"	I 621.5	BOOL	// Contagem de tucker M6 pistola 1 do DCE FAG0014
"CT_M6_01"	I 621.6	BOOL	// Contagem de tucker M6 pistola 1 do DCE FAG0014
"G0IM_G0E12_R6"	I 621.7	BOOL	// [G0IM1.G0E12]: RESERVA
"K0DPP1"	I 650.0	BOOL	// [K0TDS1.K0E11] PART 1 PRESENCE SENSOR
"K0DPP2"	I 650.1	BOOL	// [K0TDS1.K0E11] PART 5 PRESENCE SENSOR
"K0DPP3"	I 650.4	BOOL	// [K0TDS1.K0E11] PART 2 PRESENCE SENSOR
"K0DPP4"	I 650.5	BOOL	// [K0TDS1.K0E11] PART 6 PRESENCE SENSOR
"K0DPP5"	I 651.0	BOOL	// [K0TDS1.K0E11] PART 3 PRESENCE SENSOR
"K0DPP6"	I 651.1	BOOL	// [K0TDS1.K0E11] SR11 CLAMP RETURN
"K0DRSR11"	I 652.0	BOOL	// [K0TDS1.K0E11] PART 4 PRESENCE SENSOR
"K0DASR11"	I 652.1	BOOL	// [K0TDS1.K0E11] SR11 CLAMP ADVANCE
"K0DRSR12"	I 652.2	BOOL	// [K0TDS1.K0E12] SR12 CLAMP RETURN
"K0DASR12"	I 652.3	BOOL	// [K0TDS1.K0E12] SR12 CLAMP ADVANCE
"K0DRSR13"	I 652.4	BOOL	// [K0TDS1.K0E12] SR13 CLAMP RETURN
"K0DASR13"	I 652.5	BOOL	// [K0TDS1.K0E12] SR13 CLAMP ADVANCE
"K0DRSR14"	I 652.6	BOOL	// [K0TDS1.K0E12] SR14 CLAMP RETURN
"K0DASR14"	I 652.7	BOOL	// [K0TDS1.K0E12] SR14 CLAMP ADVANCE
"K0DRSR15"	I 653.0	BOOL	// [K0TDS1.K0E12] SR15 CLAMP RETURN
"K0DASR15"	I 653.1	BOOL	// [K0TDS1.K0E12] SR15 CLAMP ADVANCE
"K0DRSR16"	I 653.2	BOOL	// [K0TDS1.K0E14] SR16 CLAMP RETURN
"K0DASR16"	I 653.3	BOOL	// [K0TDS1.K0E14] SR16 CLAMP ADVANCE
"K0DRSR17"	I 653.4	BOOL	// [K0TDS1.K0E14] SR17 CLAMP RETURN
"K0DASR17"	I 653.5	BOOL	// [K0TDS1.K0E14] SR17 CLAMP ADVANCE
"K0DRSR21"	I 653.6	BOOL	// [K0TDS1.K0E13] SR21 CLAMP MANUAL RETURN
"K0DASR21"	I 653.7	BOOL	// [K0TDS1.K0E13] SR21 CLAMP MANUAL ADVANCE
"K0DRSR22"	I 654.0	BOOL	// [K0TDS1.K0E13] SR22 CLAMP MANUAL RETURN
"K0DASR22"	I 654.1	BOOL	// [K0TDS1.K0E13] SR22 CLAMP MANUAL ADVANCE
"K0DRSR23"	I 654.2	BOOL	// [K0TDS1.K0E13] SR23 CLAMP MANUAL RETURN
"K0DASR23"	I 654.3	BOOL	// [K0TDS1.K0E13] SR23 CLAMP MANUAL ADVANCE
"K0DRSR24"	I 654.4	BOOL	// [K0TDS1.K0E13] SR24 CLAMP MANUAL RETURN
"K0DASR24"	I 654.5	BOOL	// [K0TDS1.K0E13] SR24 CLAMP MANUAL ADVANCE
"K0DRSR31"	I 654.6	BOOL	// [K0TDS1.K0E13] SR31 CLAMP MANUAL RETURN
"K0DASR31"	I 654.7	BOOL	// [K0TDS1.K0E13] SR31 CLAMP MANUAL ADVANCE
"K0DRSR32"	I 655.0	BOOL	// [K0TDS1.K0E13] SR32 CLAMP MANUAL RETURN
"K0DASR32"	I 655.1	BOOL	// [K0TDS1.K0E13] SR32 CLAMP MANUAL ADVANCE
"K0_CVAL"	I 656.0	BOOL	// [K0A2] CONTRO DE COMUN SEGURIDAD
"SPARE1"	I 708.1	BOOL	// [H0TDS1.H0E15]: H0: SPARE1
"SPARE3"	I 709.2	BOOL	// [H0TDS1.H0E15]: H0: SPARE3
"SPARE5"	I 709.4	BOOL	// [H0TDS1.H0E15]: H0: SPARE5
"SPARE8"	I 709.7	BOOL	// [H0TDS1.H0E15]: H0: SPARE8
"Z2CCS1"	I 800.0	BOOL	// [Z2ZB.M02] : SAFETY COMMON 1 CONTROL (AU)
"Z2CCS2"	I 800.1	BOOL	// [Z2ZB.M02] : SAFETY COMMON 2 CONTROL (ES)
"Z2CP7b"	I 801.0	BOOL	// [Z2ZB.M03]: Z2 EV7 bar CONTROL
"Z2CRM"	I 801.1	BOOL	// [Z2ZB.M03]: Z2 CHECK GROUND CONTROL DELAY
"Z2SSZ"	I 803.2	BOOL	// [Z2ZB.M07]: Z2 ZONE SAFETY SELECTOR
"B0CCFRO1"	I 820.0	BOOL	// [B0SB.M02]: B0 F-RO1 CONTROL
"B0CCFRO2"	I 820.1	BOOL	// [B0SB.M02]: B0 F-RO2 CONTROL
"B0CCFRO3"	I 820.2	BOOL	// [B0SB.M02]: B0 F-RO3 CONTROL
"B0CCB24Z"	I 820.4	BOOL	// [B0SB.M02]: B0 CB 24V CONTROL (1-24Z)
"B0CCB24R"	I 820.5	BOOL	// [B0SB.M02]: B0 CB 24V CONTROL (2-24R)
"B0_SEL_5A"	I 821.3	BOOL
"B1BAU"	I 823.0	BOOL	// [B0SB.M08]: B1 OPERATOR 1 EGS
"B1BP1"	I 829.0	BOOL	// [B0SB.M09]: B1 T-STAND 1 BUTTON 1 (OP1) - CH1
"B1BP2"	I 829.1	BOOL	// [B0SB.M09]: B1 T-STAND 1 BUTTON 2 (OP1) - CH1
"B1BP12"	I 829.4	BOOL	// [B0SB.M09]: B1 T-STAND 1 BUTTON 1 (OP1) - CH2
"B1BP22"	I 829.5	BOOL	// [B0SB.M09]: B1 T-STAND 1 BUTTON 2 (OP1) - CH2
"Y0DDEL"	I 842.0	BOOL	// [Y0E1]: Y0: DETECTOR DESCIDA ELEVADOR
"Y0DDELH"	I 842.1	BOOL	// [Y0E1]: Y0: DETECTOR DESCIDA ELEVADOR EXTRACURSO
"Y0DPP3"	I 842.2	BOOL	// [Y0E1]: DETECTOR PRESENÇA DE PEÇA 3
"Y0E1_R1"	I 842.3	BOOL	// [Y0E1]: RESERVA
"Y0DDELPV"	I 842.4	BOOL	// [Y0E1]: Y0: DETECTOR DESCIDA ELEVADOR BAIXA VELOCIDADE
"Y0E1_R2"	I 842.5	BOOL	// [Y0E1]: RESERVA
"Y0E1_R3"	I 842.6	BOOL	// [Y0E1]: RESERVA
"Y0E1_R4"	I 842.7	BOOL	// [Y0E1]: RESERVA
"Y0DMEL"	I 843.0	BOOL	// [Y0E2]: Y0: DETECTOR SUBIDA ELEVADOR
"Y0DMELH"	I 843.1	BOOL	// [Y0E2]: Y0: DETECTOR SUBIDA ELEVADOR EXTRACURSO
"Y0DPP11"	I 843.2	BOOL	// [Y0E2]: Y0: DETECTOR PRESENÇA PEÇA 1 CH1
"Y0DPPE1"	I 843.3	BOOL	// [Y0E2]: Y0: DETECTOR PRESENÇA PEÇA ENTRADA 1
"Y0DMELPV"	I 843.4	BOOL	// [Y0E2]: Y0: DETECTOR SUBIDA ELEVADOR BAIXA VELOCIDADE
"Y0DPP2"	I 843.5	BOOL	// [Y0E2]: Y0: DETECTOR PRESENÇA PEÇA 2
"Y0DPP12"	I 843.6	BOOL	// [Y0E2]: Y0: DETECTOR PRESENÇA PEÇA 1 CH2
"Y0E2_R1"	I 843.7	BOOL	// [Y0E2]: RESERVA
"W0DPB1"	I 845.0	BOOL	// [W0E1]: CELULA PRESENÇA PEÇA B1
"W0DOB1"	I 845.1	BOOL	// [W0E1]: DETECTOR ABERTURA B1
"W0DPB2"	I 845.2	BOOL	// [W0E1]: CELULA PRESENÇA B2
"W0DOB2"	I 845.3	BOOL	// [W0E1]: DETECTOR ABERTURA B2
"W0DPB3"	I 845.4	BOOL	// [W0E1]: CELULA PRESENÇA B3
"W0DOB3"	I 845.5	BOOL	// [W0E1]: DETECTOR ABERTURA B3
"W0DP2B2"	I 845.6	BOOL	// [W0E1]: DETECTOR 2 PRESENÇA B2
"I845.7"	I 845.7	BOOL	// [W0E1]: RESERVA
"B0IFRO1"	I 846.0	BOOL	// [B0SB.M12]: B0 SAFETY COMMON 1 (FRO-1 - SC3)
"B0IFRO2"	I 847.0	BOOL	// [B0SB.M13]: B0 SAFETY COMMON 2 (FRO-2 - SC4)
"B0IFRO3"	I 848.0	BOOL	// [B0SB.M14]: B0 SAFETY COMMON 3 (FRO-3 - SC5)
"C0CCFRO1"	I 850.0	BOOL	// [C0SB.M02]: C0 F-RO1 CONTROL
"C0CCFRO2"	I 850.1	BOOL	// [C0SB.M02]: C0 F-RO2 CONTROL
"C0CCFRO3"	I 850.2	BOOL	// [C0SB.M02]: C0 F-RO3 CONTROL
"C0CCB24Z"	I 850.4	BOOL	// [C0SB.M02]: C0 CB 24V CONTROL (1-24Z)
"C0CCB24R"	I 850.5	BOOL	// [C0SB.M02]: C0 CB 24V CONTROL (2-24R)
"C1BAU"	I 853.0	BOOL	// [C0SB.M08]: C1 OPERATOR 1 EGS
"C2BAU"	I 853.1	BOOL	// [C0SB.M08]: C2 OPERATOR 2 EGS
"C1BP1"	I 859.0	BOOL	// [C0SB.M09]: B1 T-STAND 1 BUTTON 1 (OP1) - CH1
"C1BP2"	I 859.1	BOOL	// [C0SB.M09]: B1 T-STAND 1 BUTTON 2 (OP1) - CH1
"C2BP1"	I 859.2	BOOL	// [C0SB.M09]: C2 T-STAND 2 BUTTON 1 (OP2) - CH1
"C2BP2"	I 859.3	BOOL	// [C0SB.M09]: C2 T-STAND 2 BUTTON 2 (OP2) - CH1
"C1BP12"	I 859.4	BOOL	// [C0SB.M09]: B1 T-STAND 1 BUTTON 1 (OP1) - CH2
"C1BP22"	I 859.5	BOOL	// [C0SB.M09]: B1 T-STAND 1 BUTTON 2 (OP1) - CH2
"C2BP12"	I 859.6	BOOL	// [C0SB.M09]: C2 T-STAND 2 BUTTON 1 (OP2) - CH2
"C2BP22"	I 859.7	BOOL	// [C0SB.M09]: C2 T-STAND 2 BUTTON 2 (OP2) - CH2
"C0IFRO1"	I 876.0	BOOL	// [C0SB.M12]: C0 SAFETY COMMON 1 (FRO-1 - SC3)
"C0IFRO2"	I 877.0	BOOL	// [C0SB.M13]: C0 SAFETY COMMON 2 (FRO-2 - SC4)
"C0IFRO3"	I 878.0	BOOL	// [C0SB.M14]: C0 SAFETY COMMON 3 (FRO-3 - SC5)
"E0CCFRO1"	I 880.0	BOOL	// [E0SB.M02]: E0 F-RO1 CONTROL
"E0CCFRO2"	I 880.1	BOOL	// [E0SB.M02]: E0 F-RO2 CONTROL
"E0CCFRO3"	I 880.2	BOOL	// [E0SB.M02]: E0 F-RO3 CONTROL
"E0SB_M02_R1"	I 880.3	BOOL	// [E0SB.M02]: RESERVA
"E0CCB24Z"	I 880.4	BOOL	// [E0SB.M02]: E0 CB 24V CONTROL (1-24Z)
"E0CCB24R"	I 880.5	BOOL	// [E0SB.M02]: E0 CB 24V CONTROL (2-24R)
"E0SB_M02_R2"	I 880.6	BOOL	// [E0SB.M02]: RESERVA
"E0SB_M02_R3"	I 880.7	BOOL	// [E0SB.M02]: RESERVA
"E0SB_M03_R1"	I 881.0	BOOL	// [E0SB.M03]: RESERVA
"E0SB_M03_R2"	I 881.1	BOOL	// [E0SB.M03]: RESERVA
"E0SB_M03_R3"	I 881.2	BOOL	// [E0SB.M03]: RESERVA
"E0SB_M03_R4"	I 881.3	BOOL	// [E0SB.M03]: RESERVA
"E0SB_M03_R5"	I 881.4	BOOL	// [E0SB.M03]: RESERVA
"E0SB_M03_R6"	I 881.5	BOOL	// [E0SB.M03]: RESERVA
"E0SB_M03_R7"	I 881.6	BOOL	// [E0SB.M03]: RESERVA
"E0SB_M03_R8"	I 881.7	BOOL	// [E0SB.M03]: RESERVA
"E1BAU"	I 883.0	BOOL	// [E0SB.M08]: E1 OPERATOR 1 EGS
"E2BAU"	I 883.1	BOOL	// [E0SB.M08]: E2 OPERATOR 2 EGS
"E0SB_M08_R1"	I 883.2	BOOL	// [E0SB.M08]: RESERVA
"E0SB_M08_R2"	I 883.3	BOOL	// [E0SB.M08]: RESERVA
"E1BP1"	I 889.0	BOOL	// [E0SB.M09]: E1 T-STAND 1 BUTTON 1 (OP1) - CH1
"E1BP2"	I 889.1	BOOL	// [E0SB.M09]: E1 T-STAND 1 BUTTON 2 (OP1) - CH1
"E2BP1"	I 889.2	BOOL	// [E0SB.M09]: E2 T-STAND 2 BUTTON 1 (OP2) - CH1
"E2BP2"	I 889.3	BOOL	// [E0SB.M09]: E2 T-STAND 2 BUTTON 2 (OP2) - CH1
"E1BP12"	I 889.4	BOOL	// [E0SB.M09]: E1 T-STAND 1 BUTTON 1 (OP1) - CH2
"E1BP22"	I 889.5	BOOL	// [E0SB.M09]: E1 T-STAND 1 BUTTON 2 (OP1) - CH2
"E2BP12"	I 889.6	BOOL	// [E0SB.M09]: E2 T-STAND 2 BUTTON 1 (OP2) - CH2
"E2BP22"	I 889.7	BOOL	// [E0SB.M09]: E2 T-STAND 2 BUTTON 2 (OP2) - CH2
"E1CPOP1"	I 895.0	BOOL	// [E0SB.M10]: LASER SCANNER 1 CH1
"E2CPOP1"	I 895.2	BOOL	// [E0SB.M10]: LASER SCANNER 2 CH1
"E1CPOP2"	I 895.4	BOOL	// [E0SB.M10]: LASER SCANNER 1 CH2
"E2CPOP2"	I 895.6	BOOL	// [E0SB.M10]: LASER SCANNER 2 CH2
"E0IFRO1"	I 906.0	BOOL	// [E0SB.M12]: E0 SAFETY COMMON 1 (FRO-1 - SC3)
"E0IFRO2"	I 907.0	BOOL	// [E0SB.M13]: E0 SAFETY COMMON 2 (FRO-2 - SC4)
"E0IFRO3"	I 908.0	BOOL	// [E0SB.M14]: E0 SAFETY COMMON 3 (FRO-3 - SC5)
"G0CCFRO1"	I 910.0	BOOL	// [G0SB.M02]: G0 F-RO1 CONTROL
"G0CCFRO2"	I 910.1	BOOL	// [G0SB.M02]: G0 F-RO2 CONTROL
"G0CCFRO3"	I 910.2	BOOL	// [G0SB.M02]: G0 F-RO3 CONTROL
"J0DPP1"	I 910.3	BOOL	// [J0OPB.M2] Detector presencia de pieza 1
"G0CCB24Z"	I 910.4	BOOL	// [G0SB.M02]: G0 CB 24V CONTROL (1-24Z)
"G0CCB24R"	I 910.5	BOOL	// [G0SB.M02]: G0 CB 24V CONTROL (2-24R)
"J0OP11VAL"	I 910.6	BOOL	// [J0OPB:M3] OPERADOR 1 CONTACTO 1
"J0OP12VAL"	I 910.7	BOOL	// [J0OPB:M3] OPERADOR 1 CONTACTO 2
"G0SB_M03_R1"	I 911.0	BOOL	// [G0SB.M03]: RESERVA
"G0SB_M03_R2"	I 911.1	BOOL	// [G0SB.M03]: RESERVA
"G0SB_M03_R3"	I 911.2	BOOL	// [G0SB.M03]: RESERVA
"G0SB_M03_R4"	I 911.3	BOOL	// [G0SB.M03]: RESERVA
"G0SB_M03_R6"	I 911.5	BOOL	// [G0SB.M03]: RESERVA
"G0SB_M03_R8"	I 911.7	BOOL	// [G0SB.M03]: RESERVA
"G0SB_M08_R1"	I 912.2	BOOL	// [G0SB.M08]: RESERVA
"G0SB_M08_R2"	I 912.3	BOOL	// [G0SB.M08]: RESERVA
"G1BAU"	I 913.0	BOOL	// [G0SB.M08]: G1 OPERATOR 1 EGS
"G2BAU"	I 913.1	BOOL	// [G0SB.M08]: G2 OPERATOR 2 EGS
"G1BP1"	I 919.0	BOOL	// [G0SB.M09]: G1 T-STAND 1 BUTTON 1 (OP1) - CH1
"G1BP2"	I 919.1	BOOL	// [G0SB.M09]: G1 T-STAND 1 BUTTON 2 (OP1) - CH1
"G2BP1"	I 919.2	BOOL	// [G0SB.M09]: G2 T-STAND 2 BUTTON 1 (OP2) - CH1
"G2BP2"	I 919.3	BOOL	// [G0SB.M09]: G2 T-STAND 2 BUTTON 2 (OP2) - CH1
"G1BP12"	I 919.4	BOOL	// [G0SB.M09]: G1 T-STAND 1 BUTTON 1 (OP1) - CH2
"G1BP22"	I 919.5	BOOL	// [G0SB.M09]: G1 T-STAND 1 BUTTON 2 (OP1) - CH2
"G2BP12"	I 919.6	BOOL	// [G0SB.M09]: G2 T-STAND 2 BUTTON 1 (OP2) - CH2
"G2BP22"	I 919.7	BOOL	// [G0SB.M09]: G2 T-STAND 2 BUTTON 2 (OP2) - CH2
"G0SB_M10_R1"	I 924.0	BOOL	// [G0SB.M10]: RESERVA
"G0SB_M10_R2"	I 924.1	BOOL	// [G0SB.M10]: RESERVA
"G0SB_M10_R3"	I 924.2	BOOL	// [G0SB.M10]: RESERVA
"G0SB_M10_R4"	I 924.3	BOOL	// [G0SB.M10]: RESERVA
"G0IFRO1"	I 935.0	BOOL	// [G0SB.M12]: G0 SAFETY COMMON 1 (FRO-1 - SC3)
"G0IFRO2"	I 936.0	BOOL	// [G0SB.M13]: G0 SAFETY COMMON 2 (FRO-2 - SC4)
"G0IFRO3"	I 937.0	BOOL	// [G0SB.M14]: G0 SAFETY COMMON 3 (FRO-3 - SC5)
"J0CCB24Z"	I 940.4	BOOL	// [J0OPB.M02]: C0 CB 24V CONTROL (1-24Z)
"J0CCB24R"	I 940.5	BOOL	// [J0OPB.M02]: C0 CB 24V CONTROL (2-24R)
"B0DRPL1"	I 950.0	BOOL	// [B0TDS1.B0E1]: B0: DETECTOR RETROCESO PL1
"B0DAPL1"	I 950.1	BOOL	// [B0TDS1.B0E1]: B0: DETECTOR AVANCE PL1
"B0DRSR2"	I 950.2	BOOL	// [B0TDS1.B0E1]: B0: DETECTOR RETROCESO SR2
"B0DASR2"	I 950.3	BOOL	// [B0TDS1.B0E1]: B0: DETECTOR AVANCE SR2
"B0DRSR3"	I 950.4	BOOL	// [B0TDS1.B0E1]: B0: DETECTOR RETROCESO SR3
"B0DASR3"	I 950.5	BOOL	// [B0TDS1.B0E1]: B0: DETECTOR AVANCE SR3
"B0DPP1"	I 951.0	BOOL	// [B0TDS1.B0E1]: B0: DETECTOR PRESENCIA DE PIEZA 1
"B0DPP2"	I 951.2	BOOL	// [B0TDS1.B0E1]: B0: DETECTOR PRESENCIA DE PIEZA 2
"B0DPP3"	I 951.4	BOOL	// [B0TDS1.B0E1]: B0: DETECTOR PRESENCIA DE PIEZA 3
"C0DRPL1"	I 960.0	BOOL	// [C0TDS1.C0E1]: C0: DETECTOR RETROCESO PL1
"C0DAPL1"	I 960.1	BOOL	// [C0TDS1.C0E1]: C0: DETECTOR AVANCE PL1
"C0DRSR2"	I 960.2	BOOL	// [C0TDS1.C0E1]: C0: DETECTOR RETROCESO SR2
"C0DASR2"	I 960.3	BOOL	// [C0TDS1.C0E1]: C0: DETECTOR AVANCE SR2
"C0DRSR3"	I 960.4	BOOL	// [C0TDS1.C0E1]: C0: DETECTOR RETROCESO SR3
"C0DASR3"	I 960.5	BOOL	// [C0TDS1.C0E1]: C0: DETECTOR AVANCE SR3
"C0DPP1"	I 961.4	BOOL	// [C0TDS1.C0E1]: C0: DETECTOR PRESENCIA DE PIEZA 1
"E0DRSR1"	I 1040.0	BOOL	// [E0TDS1.E0E1]: E0: DETECTOR RETROCESO SR1
"E0DASR1"	I 1040.1	BOOL	// [E0TDS1.E0E1]: E0: DETECTOR AVANCE SR1
"E0DRSR2"	I 1040.2	BOOL	// [E0TDS1.E0E1]: E0: DETECTOR RETROCESO SR2
"E0DASR2"	I 1040.3	BOOL	// [E0TDS1.E0E1]: E0: DETECTOR AVANCE SR2
"E0DRSR3"	I 1040.4	BOOL	// [E0TDS1.E0E1]: E0: DETECTOR RETROCESO SR3
"E0DASR3"	I 1040.5	BOOL	// [E0TDS1.E0E1]: E0: DETECTOR AVANCE SR3
"E0DRVU4"	I 1040.6	BOOL	// [E0TDS1.E0E1]: E0: DETECTOR RETROCESO VU4
"E0DAVU4"	I 1040.7	BOOL	// [E0TDS1.E0E1]: E0: DETECTOR AVANCE VU4
"E0DRVU5"	I 1041.0	BOOL	// [E0TDS1.E0E1]: E0: DETECTOR RETROCESO VU5
"E0DAVU5"	I 1041.1	BOOL	// [E0TDS1.E0E1]: E0: DETECTOR AVANCE VU5
"E0DRSR6"	I 1041.2	BOOL	// [E0TDS1.E0E1]: E0: DETECTOR RETROCESO SR6
"E0DASR6"	I 1041.3	BOOL	// [E0TDS1.E0E1]: E0: DETECTOR AVANCE SR6
"E0DPPX675A"	I 1041.4	BOOL	// [E0TDS1.E0E1]: E0: DETECTOR PRESENCIA PIEZA CASOLETA 5 ASIENTOS
"E0DPPX672A"	I 1041.5	BOOL	// [E0TDS1.E0E1]: E0: DETECTOR AUSCENCIA PIEZA CASOLETA 5 ASIENTOS
"E0DPP1"	I 1041.6	BOOL	// [E0TDS1.E0E1]: E0: DETECTOR PIEZA 1
"G0DRSR1"	I 1060.0	BOOL	// [G0TDS1.G0E1]: G0: DETECTOR RETROCESO SR1
"G0DASR1"	I 1060.1	BOOL	// [G0TDS1.G0E1]: G0: DETECTOR AVANCE SR1
"G0DRSR2"	I 1060.2	BOOL	// [G0TDS1.G0E1]: G0: DETECTOR RETROCESO SR2
"G0DASR2"	I 1060.3	BOOL	// [G0TDS1.G0E1]: G0: DETECTOR AVANCE SR2
"G0DRSR3"	I 1060.4	BOOL	// [G0TDS1.G0E1]: G0: DETECTOR RETROCESO SR3
"G0DASR3"	I 1060.5	BOOL	// [G0TDS1.G0E1]: G0: DETECTOR AVANCE SR3
"G0DPP1"	I 1061.0	BOOL	// [G0TDS1.E01]: G0: DETECTOR PRESENCIA PIEZA  1
"G0DPP2"	I 1061.2	BOOL	// [G0TDS1.E01]: G0: DETECTOR PRESENCIA PIEZA  2
"L0DAPS11"	I 1070.0	BOOL	// L0: Sensor avance PIN SHIFT 1-1
"L0DRPS11"	I 1070.1	BOOL	// L0: Sensor retroceso PIN SHIFT 1-1
"L0DAPS12"	I 1070.2	BOOL	// L0: Sensor avance PIN SHIFT 1-2
"L0DRPS12"	I 1070.3	BOOL	// L0: Sensor retroceso PIN SHIFT 1-2
"L0DAPS13"	I 1070.4	BOOL	// L0: Sensor avance PIN SHIFT 1-3
"L0DRPS13"	I 1070.5	BOOL	// L0: Sensor retroceso PIN SHIFT 1-3
"L0DAPS14"	I 1070.6	BOOL	// L0: Sensor avance PIN SHIFT 1-4
"L0DRPS14"	I 1070.7	BOOL	// L0: Sensor retroceso PIN SHIFT 1-4
"L0DASR11"	I 1071.0	BOOL	// L0: Sensor avance CLAMP 1-1
"L0DRSR11"	I 1071.1	BOOL	// L0: Sensor retroceso CLAMP 1-1
"L0DASR12"	I 1071.2	BOOL	// L0: Sensor avance CLAMP 1-2
"L0DRSR12"	I 1071.3	BOOL	// L0: Sensor retroceso CLAMP 1-2
"L0DASR13"	I 1071.4	BOOL	// L0: Sensor avance CLAMP 1-3
"L0DRSR13"	I 1071.5	BOOL	// L0: Sensor retroceso CLAMP 1-3
"L0DASR14"	I 1071.6	BOOL	// L0: Sensor avance CLAMP 1-4
"L0DRSR14"	I 1071.7	BOOL	// L0: Sensor retroceso CLAMP 1-4
"L0DASR21"	I 1072.0	BOOL	// L0: Sensor avance CLAMP 2-1
"L0DRSR21"	I 1072.1	BOOL	// L0: Sensor retroceso CLAMP 2-1
"L0DASR22"	I 1072.2	BOOL	// L0: Sensor avance CLAMP 2-2
"L0DRSR22"	I 1072.3	BOOL	// L0: Sensor retroceso CLAMP 2-2
"L0DASR23"	I 1072.4	BOOL	// L0: Sensor avance CLAMP 2-3
"L0DRSR23"	I 1072.5	BOOL	// L0: Sensor retroceso CLAMP 2-3
"L0DASR41"	I 1072.6	BOOL	// L0: Sensor avance CLAMP 4-1
"L0DRSR41"	I 1072.7	BOOL	// L0: Sensor retroceso CLAMP 4-2
"L0DASR25"	I 1073.0	BOOL	// L0: Sensor avance CLAMP 2-5
"L0DRSR25"	I 1073.1	BOOL	// L0: Sensor retroceso CLAMP 2-5
"L0DASR31"	I 1073.2	BOOL	// L0: Sensor avance HAND CLAMP 3-1
"L0DRSR31"	I 1073.3	BOOL	// L0: Sensor retroceso HAND CLAMP 3-1
"L0DAVU11"	I 1073.4	BOOL	// L0: Sensor avance EJECTOR 1-1
"L0DRVU11"	I 1073.5	BOOL	// L0: Sensor retroceso  EJECTOR 1-1
"L0DAVU12"	I 1073.6	BOOL	// L0: Sensor avance EJECTOR 1-2
"L0DRVU12"	I 1073.7	BOOL	// L0: Sensor retroceso  EJECTOR 1-2
"L0DAVU13"	I 1074.0	BOOL	// L0: Sensor avance EJECTOR 1-3
"L0DRVU13"	I 1074.1	BOOL	// L0: Sensor retroceso EJECTOR 1-3
"L0DAVU21"	I 1074.2	BOOL	// L0: Sensor avance PINGYI 2-1
"L0DRVU21"	I 1074.3	BOOL	// L0: Sensor retroceso PINGYI 2-1
"L0DAVU22"	I 1074.4	BOOL	// L0: Sensor avance PINGYI 2-2
"L0DRVU22"	I 1074.5	BOOL	// L0: Sensor retroceso PINGYI 2-2
"L0DAVU23"	I 1074.6	BOOL	// L0: Sensor avance PINGYI 2-3
"L0DRVU23"	I 1074.7	BOOL	// L0: Sensor retroceso PINGYI 2-3
"L0DAVU24"	I 1075.0	BOOL	// L0: Sensor avance PINGYI 2-4
"L0DRVU24"	I 1075.1	BOOL	// L0: Sensor retroceso PINGYI 2-4
"L0DPP1"	I 1075.4	BOOL	// Detector precencia 1
"L0DPP2"	I 1075.5	BOOL	// Detector precencia 2
"L0DPP3"	I 1075.6	BOOL	// Detector precencia 3
"L0DPP4"	I 1075.7	BOOL	// Detector precencia 4
"L0DPP5"	I 1076.0	BOOL	// Detector precencia 5
"L0DPP6"	I 1076.1	BOOL	// Detector precencia 6
"L0DPP7"	I 1076.2	BOOL	// Detector precencia 7
"L0DPP8"	I 1076.3	BOOL	// Detector precencia 8
"L0DPP9"	I 1076.4	BOOL	// Detector precencia 9
"L0DPP10"	I 1076.5	BOOL	// Detector precencia 10
"L0DPP11"	I 1076.6	BOOL	// Detector precencia 11
"L0DPP12"	I 1076.7	BOOL	// Detector precencia 12
"L0DPP13"	I 1077.0	BOOL	// Detector precencia 13
"L0DPP14"	I 1077.1	BOOL	// Detector precencia 14
"L0DPP15"	I 1077.2	BOOL	// Detector precencia 15
"L1BROC"	I 1078.6	BOOL	// L1: PULSADOR RETORNO A ORIGEN
"L0DPVO1"	I 1079.6	BOOL	//  L0IM1 PRESSURE SWITCH
"L1BAU1"	I 1080.0	BOOL	// Festo parada de emergencia 11 L0
"L1BP1"	I 1080.1	BOOL	// Festo bimanual 11 L0
"L2BAU1"	I 1080.2	BOOL	// Festo parada de emergencia 21 L0
"L2BP1"	I 1080.3	BOOL	// Festo bimanual 21 L0
"L1BAU2"	I 1080.4	BOOL	// Festo parada de emergencia 12 L0
"L1BP2"	I 1080.5	BOOL	// Festo bimanual 12 L0
"L2BAU2"	I 1080.6	BOOL	// Festo parada de emergencia 22 L0
"L2BP2"	I 1080.7	BOOL	// Festo bimanual 22 L0
"L0CCSOP"	I 1087.0	BOOL	// L0IM1: CONTROL DE CANAL
"M0DASR11"	I 1100.0	BOOL	// M0: Sensor avance HAND CLAMP 1-1
"M0DRSR11"	I 1100.1	BOOL	// M0: Sensor retroceso HAND CLAMP 1-1
"M0DASR12"	I 1100.2	BOOL	// M0: Sensor avance HAND CLAMP 1-2
"M0DRSR12"	I 1100.3	BOOL	// M0: Sensor retroceso HAND CLAMP 1-2
"M0DASR21"	I 1100.4	BOOL	// M0: Sensor avance CLAMP 2-1
"M0DRSR21"	I 1100.5	BOOL	// M0: Sensor retroceso CLAMP 2-1
"M0DASR22"	I 1100.6	BOOL	// M0: Sensor avance CLAMP 2-2
"M0DRSR22"	I 1100.7	BOOL	// M0: Sensor retroceso CLAMP 2-2
"M0DAVU11"	I 1101.0	BOOL	// M0: Sensor avance EJECTOR 1-1
"M0DRVU11"	I 1101.1	BOOL	// M0: Sensor retroceso EJECTOR 1-1
"M0DAVU12"	I 1101.2	BOOL	// M0: Sensor avance EJECTOR 1-2
"M0DRVU12"	I 1101.3	BOOL	// M0: Sensor retroceso EJECTOR 1-2
"M0DAVU13"	I 1101.4	BOOL	// M0: Sensor avance EJECTOR 1-3
"M0DRVU13"	I 1101.5	BOOL	// M0: Sensor retroceso EJECTOR 1-3
"M0DAVU14"	I 1101.6	BOOL	// M0: Sensor avance EJECTOR 1-4
"M0DRVU14"	I 1101.7	BOOL	// M0: Sensor retroceso EJECTOR 1-4
"M0DPP1"	I 1102.0	BOOL	//  M0: Detector de presencia 1
"M0DPP2"	I 1102.1	BOOL	//  M0: Detector de presencia 2
"M0DPP3"	I 1102.2	BOOL	//  M0: Detector de presencia 3
"M0DPP4"	I 1102.3	BOOL	//  M0: Detector de presencia 4
"M0DPP5"	I 1102.4	BOOL	//  M0: Detector de presencia 5
"M0DPP6"	I 1102.5	BOOL	//  M0: Detector de presencia 6
"M1BROC"	I 1103.0	BOOL	//  M1: BOTON RETORNO AL ORIGEN
"M0DPVO1"	I 1103.6	BOOL	//  M0IM1 PRESSURE SWITCH
"M1BAU1"	I 1104.0	BOOL	// FESTO parada de emergencia M11
"M1BP1"	I 1104.1	BOOL	// FESTO boton bimanual M11
"M2BAU1"	I 1104.2	BOOL	// FESTO parada de emergencia M21
"M2BP1"	I 1104.3	BOOL	// FESTO boton bimanual M21
"M1BAU2"	I 1104.4	BOOL	// FESTO parada de emergencia M12
"M1BP2"	I 1104.5	BOOL	// FESTO boton bimanual M12
"M2BAU2"	I 1104.6	BOOL	// FESTO parada de emergencia M22
"M2BP2"	I 1104.7	BOOL	// FESTO boton bimanual M22
"M0CCSOP"	I 1111.0	BOOL	// M0IM1: CONTROL CANAL 0
"N0DRPLA1"	I 1150.0	BOOL
"N0DAPLA1"	I 1150.1	BOOL
"N0DRPLA2"	I 1150.2	BOOL
"N0DAPLA2"	I 1150.3	BOOL
"N0DRPLA3"	I 1150.4	BOOL
"N0DAPLA3"	I 1150.5	BOOL
"N0DRPLA4"	I 1150.6	BOOL
"N0DAPLA4"	I 1150.7	BOOL
"N0DRCLB1"	I 1151.0	BOOL
"N0DACLB1"	I 1151.1	BOOL
"N0DRPLC1"	I 1151.2	BOOL
"N0DAPLC1"	I 1151.3	BOOL
"N0DRPLC2"	I 1151.4	BOOL
"N0DAPLC2"	I 1151.5	BOOL
"N0DRSRD1"	I 1151.6	BOOL
"N0DASRD1"	I 1151.7	BOOL
"N0DRSRD2"	I 1152.0	BOOL
"N0DASRD2"	I 1152.1	BOOL
"N0DRSRE1"	I 1152.2	BOOL
"N0DASRE1"	I 1152.3	BOOL
"N0DRSRE2"	I 1152.4	BOOL
"N0DASRE2"	I 1152.5	BOOL
"N0DRSRF1"	I 1152.6	BOOL
"N0DASRF1"	I 1152.7	BOOL
"N0DRSRF2"	I 1153.0	BOOL
"N0DASRF2"	I 1153.1	BOOL
"N0DRSRF3"	I 1153.2	BOOL
"N0DASRF3"	I 1153.3	BOOL
"N0DRSRF4"	I 1153.4	BOOL
"N0DASRF4"	I 1153.5	BOOL
"N0DRSRF5"	I 1153.6	BOOL
"N0DASRF5"	I 1153.7	BOOL
"N0DRSRF6"	I 1154.0	BOOL
"N0DASRF6"	I 1154.1	BOOL
"N0DRCLG1"	I 1154.2	BOOL
"N0DACLG1"	I 1154.3	BOOL
"N0DRCLH1"	I 1154.4	BOOL
"N0DACLH1"	I 1154.5	BOOL
"N0DRSRJ1"	I 1154.6	BOOL
"N0DASRJ1"	I 1154.7	BOOL
"N0DRSRJ2"	I 1155.0	BOOL
"N0DASRJ2"	I 1155.1	BOOL
"N0DRCLK1"	I 1155.2	BOOL
"N0DACLK1"	I 1155.3	BOOL
"N0DACLK2"	I 1155.4	BOOL
"N0_SEL_LB"	I 1155.6	BOOL	// N0IM1: SELECTOR DE MODELO L/B
"N0DPP1"	I 1156.0	BOOL	// DETECTOR PRESENCIA DE PIEZA 1
"N0DPP3"	I 1156.1	BOOL	// DETECTOR PRESENCIA DE PIEZA 2
"N0DPP7"	I 1156.2	BOOL	// DETECTOR PRESENCIA DE PIEZA 4
"N0DPP5"	I 1156.3	BOOL	// DETECTOR PRESENCIA DE PIEZA 3
"N0DPP4"	I 1156.4	BOOL	// DETECTOR PRESENCIA DE PIEZA 6
"N0DPP2"	I 1156.5	BOOL	// DETECTOR PRESENCIA DE PIEZA 5
"N0DPP6"	I 1156.6	BOOL	// DETECTOR PRESENCIA DE PIEZA 7
"N0DPP8"	I 1156.7	BOOL	// DETECTOR PRESENCIA DE PIEZA 8
"N0DPP9"	I 1157.0	BOOL	// DETECTOR PRESENCIA DE PIEZA 9
"N0DPP10"	I 1157.2	BOOL	// DETECTOR PRESENCIA DE PIEZA 10
"N0DPP11"	I 1157.4	BOOL	// DETECTOR PRESENCIA DE PIEZA 11
"INFO_MANT"	I 1157.5	BOOL	// VARIABLE MODO MANTENIMIENTO
"N0CP7B"	I 1157.6	BOOL	// PRESOSTATO
"N0BAU1"	I 1158.0	BOOL	// FESTO parada de emergencia N11
"N0_BI11"	I 1158.1	BOOL	// FESTO boton bimanual N11
"N0_BAU2"	I 1158.2	BOOL	// FESTO parada de emergencia N21
"N0_BI21"	I 1158.3	BOOL	// FESTO boton bimanual N21
"N0_BAU12"	I 1158.4	BOOL	// FESTO parada de emergencia N12
"N0_BI12"	I 1158.5	BOOL	// FESTO boton bimanual N12
"N0_BAU22"	I 1158.6	BOOL	// FESTO parada de emergencia N22
"N0_BI22"	I 1158.7	BOOL	// FESTO boton bimanual N22
"N0CCSOP"	I 1165.0	BOOL	// N0IM1: CONTROL CANAL 0
"E0DPVR"	I 2803.3	BOOL	// [E0SB.G120D]: E0 DETECTOR DE PEQUEÑA VELOCIDAD RETROCESO
"E0DPVA"	I 2803.4	BOOL	// [E0SB.G120D]: E0 DETECTOR DE PEQUEÑA VELOCIDAD AVANCE
"RES1"	I 2803.5	BOOL
"E0DDP1"	I 2803.6	BOOL	// [E0SB.G120D]: E0 DETECTOR DE SOBREPASO 1
"E0DPOS180"	I 2947.0	BOOL	// [E0SB.G120D]: E0 DETECTOR DE POSICION 180º
"E0DPOS0"	I 2947.2	BOOL	// [E0SB.G120D]: E0 DETECTOR DE POSICION 0º
"E0DPOS90"	I 2947.3	BOOL	// [E0SB.G120D]: E0 DETECTOR DE POSICION 90º
"BA0"	M 0.0	BOOL	// FACILITY: BIT ALWAYS OFF / ILOT: BIT TOUJOURS A 0
"BA1"	M 0.1	BOOL	// FACILITY: BIT ALWAYS ON / ILOT: BIT TOUJOURS A 1
"BA1LIEN"	M 0.2	BOOL	// FACILITY: BIT ALWAYS ON (LINK IN THE PROGRAMMING NETWORK)
"SHUNT"	M 0.3	BOOL	// BIT FOR BYPASS DURING FACILITY START UP / BIT SHUNT POUR LA MISE AU POINT
"PERSO"	M 0.4	BOOL	// NEED TO PERSONALIZE BY THE PROGRAMMER / EQUATION A PERSONNALISER
"POUB"	M 0.5	BOOL	// DUST BIN BIT / BIT POUBELLE
"Temp_Z2"	M 0.6	BOOL	// bit especial nueva zona 2
"SYSFROID"	M 0.7	BOOL	// DETECTING COLD START PLC (OB102) / DETECTION DEMARRAGE A FROID API (OB102)
"ICL040S"	M 1.2	BOOL	// BLINKING INFORMATION / INFORMATION CLIGNOTEMENT
"ICL080S"	M 1.4	BOOL	// BLINKING INFORMATION / INFORMATION CLIGNOTEMENT
"ICL2S"	M 1.7	BOOL	// BLINKING INFORMATION / INFORMATION CLIGNOTEMENT
"Z3kau"	M 4.0	BOOL
"Z3CCAU"	M 4.1	BOOL
"Z3CFROAU"	M 4.2	BOOL
"B0BPSVAL_X1"	M 5.0	BOOL	// BOTÃO DE BYPASS POSSIBILIDADE 1 - IHM
"B0BPVAL_X2"	M 5.1	BOOL	// BOTÃO BYPASS POSSIBILIDADE 2 - IHM
"SEL_GIRO"	M 9.0	BOOL	// SELECCIO DE GIRO: 0=2 POS; 1=4 POS
"IADF"	M 10.1	BOOL	// FACILITY: FAULT RESET INFORMATION (SAFETY)
"IR"	M 10.2	BOOL	// FACILITY: CONTROL ON INFORMATION (SAFETY)
"SHUNT_ADAMI"	M 10.7	BOOL
"Z1DEF_MAJ"	M 11.0	BOOL	// ZONE 1: MAJOR FAULT (SAFETY)
"Z1IADF"	M 11.1	BOOL	// ZONE 1: FAULT RESET INFORMATION (SAFETY)
"Z1IR"	M 11.2	BOOL	// ZONE 1: CONTROL ON INFORMATION (SAFETY)
"Z1IAFJ"	M 11.3	BOOL	// ZONE 1: END OF PRODUCTION STOP INFORMATION (SAFETY)
"Z8DEF_MAJ"	M 11.4	BOOL	// ZONE 8: MAJOR FAULT (SAFETY)
"Z8IADF"	M 11.5	BOOL	// ZONE 8: FAULT RESET INFORMATION (SAFETY)
"Z8IR"	M 11.6	BOOL	// ZONE 8: CONTROL ON INFORMATION (SAFETY)
"Z8IAFJ"	M 11.7	BOOL	// ZONE 8: END OF PRODUCTION STOP INFORMATION (SAFETY)
"SELETTRA"	M 12.0	BOOL	// PRECISA FAZER VERIFICAÇÃO
"Z3def_maj"	M 12.1	BOOL
"Z3Ir"	M 12.2	BOOL
"Z3MAUTO"	M 12.3	BOOL
"Z3MANU"	M 12.4	BOOL
"Z3Iadf"	M 12.5	BOOL
"A1DINHIB1"	M 15.0	BOOL	// A1 DEMANDA DE MODIFICACION DE SEGURIDAD
"A2DINHIB1"	M 15.1	BOOL	// A2 DEMANDA DE MODIFICACION DE SEGURIDAD
"A3DINHIB1"	M 15.2	BOOL	// A3 DEMANDA DE MODIFICACION DE SEGURIDAD
"A4DINHIB1"	M 15.3	BOOL	// A4 DEMANDA DE MODIFICACION DE SEGURIDAD
"D1DINHIB1"	M 15.4	BOOL	// D1 DEMANDA DE MODIFICACION DE SEGURIDAD
"D2DINHIB1"	M 15.5	BOOL	// D2 DEMANDA DE MODIFICACION DE SEGURIDAD
"D3DINHIB1"	M 15.6	BOOL	// D3 DEMANDA DE MODIFICACION DE SEGURIDAD
"D4DINHIB1"	M 15.7	BOOL	// D4 DEMANDA DE MODIFICACION DE SEGURIDAD
"F1DINHIB1"	M 16.0	BOOL	// F1 DEMANDA DE MODIFICACION DE SEGURIDAD
"F2DINHIB1"	M 16.1	BOOL	// F2 DEMANDA DE MODIFICACION DE SEGURIDAD
"DEFMAJ_AU_ES"	M 16.5	BOOL
"Z3IAFJ"	M 18.0	BOOL
"Z2DEF_MAJ"	M 21.0	BOOL	// ZONE 2: MAJOR FAULT (SAFETY)
"Z2IADF"	M 21.1	BOOL	// ZONE 2: CONTROL ON INFORMATION (SAFETY)
"Z2IR"	M 21.2	BOOL	// ZONE 2: END OF PRODUCTION STOP INFORMATION (SAFETY)
"Z2IAFJ"	M 21.3	BOOL	// ZONE 2: END OF PRODUCTION STOP INFORMATION (SAFETY)
"SHUNT_ADAMI_SFMF"	M 29.0	BOOL
"H_D0PLE_AUT"	M 30.0	BOOL	// Habilitação PLE avanço automatico
"D0_XAA"	M 30.1	BOOL	// D0: Auxiliar autorização de avanço PLE
"H_A0PLE_AUT"	M 30.2	BOOL	// Habilitação avanço PLE automatico A0
"A0_XAAPLE"	M 30.3	BOOL	// Auxiliar autorização avanço A0
"MCFPY"	M 40.0	BOOL	// Memoria Condição de Falha Poka Yoke Mesa D0
"xAlas"	M 41.0	BOOL	//  alarma sonora y luminosa MOP
"A0.DEF"	M 42.0	BOOL	// DEFECTO MESA A0
"D0.DEF"	M 42.1	BOOL	// DEFECTO MESA D0
"F0.DEF"	M 42.2	BOOL	//  DEFECTO MESA
"SEL_x67_2A"	M 50.0	BOOL
"SHUNT_CRUZETA_D0"	M 95.1	BOOL
"SHUNT_CRUZETA_F0"	M 95.2	BOOL
"C2VINHIB"	M 97.0	BOOL	// G2 VALIDACION DE MODIFICACION DE SEGURIDAD
"C2SOPVINH"	M 97.1	BOOL	// G2 LAMPADA SEGURIDAD INACTIVO
"C2MINHIB"	M 97.2	BOOL	// G2 MEMORIA INHIBICION DE SEGURIDAD
"C2ACONF"	M 98.0	BOOL	// G2 AUTHORIZACION DE MODIFICACION DE SEGURIDAD
"C2DINHIB1"	M 98.1	BOOL	// G2 DEMANDA DE MODIFICACION DE SEGURIDAD 1
"C1ACONF"	M 98.3	BOOL	// G1 AUTHORIZACION DE MODIFICACION DE SEGURIDAD
"C1VINHIB"	M 98.4	BOOL	// G1 VALIDACION DE MODIFICACION DE SEGURIDAD
"C1SOPVINH"	M 98.5	BOOL	// G1 LAMPADA SEGURIDAD INACTIVO
"C1MINHIB"	M 98.6	BOOL	// G1 MEMORIA INHIBICION DE SEGURIDAD
"C1DINHIB1"	M 98.7	BOOL	// G1 DEMANDA DE MODIFICACION DE SEGURIDAD 1
"G2ACONF"	M 99.0	BOOL	// G2 AUTHORIZACION DE MODIFICACION DE SEGURIDAD
"G2DINHIB1"	M 99.1	BOOL	// G2 DEMANDA DE MODIFICACION DE SEGURIDAD 1
"E2ACONF"	M 99.2	BOOL	// E2 AUTHORIZACION DE MODIFICACION DE SEGURIDAD
"E2DINHIB1"	M 99.3	BOOL	// E2 DEMANDA DE MODIFICACION DE SEGURIDAD 1
"ANALISAR"	M 100.2	BOOL	// ANALISAR DEPOIS
"PLANO_A"	M 100.5	BOOL	// HABILITA BARCODE
"E1DINHIB1"	M 101.0	BOOL	// E1 DEMANDA DE MODIFICACION DE SEGURIDAD 1
"E2VINHIB"	M 102.0	BOOL	// E2 VALIDACION DE MODIFICACION DE SEGURIDAD
"E2SOPVINH"	M 102.1	BOOL	// E2 LAMPADA SEGURIDAD INACTIVO
"E2MINHIB"	M 102.2	BOOL	// E2 MEMORIA INHIBICION DE SEGURIDAD
"E1ACONF"	M 102.3	BOOL	// E1 AUTHORIZACION DE MODIFICACION DE SEGURIDAD
"E1VINHIB"	M 102.4	BOOL	// E1 VALIDACION DE MODIFICACION DE SEGURIDAD
"E1SOPVINH"	M 102.5	BOOL	// E1 LAMPADA SEGURIDAD INACTIVO
"E1MINHIB"	M 102.6	BOOL	// E1 MEMORIA INHIBICION DE SEGURIDAD
"G1DINHIB1"	M 102.7	BOOL	// G1 DEMANDA DE MODIFICACION DE SEGURIDAD 1
"G2VINHIB"	M 103.0	BOOL	// G2 VALIDACION DE MODIFICACION DE SEGURIDAD
"G2SOPVINH"	M 103.1	BOOL	// G2 LAMPADA SEGURIDAD INACTIVO
"G2MINHIB"	M 103.2	BOOL	// G2 MEMORIA INHIBICION DE SEGURIDAD
"G1ACONF"	M 103.3	BOOL	// G1 AUTHORIZACION DE MODIFICACION DE SEGURIDAD
"G1VINHIB"	M 103.4	BOOL	// G1 VALIDACION DE MODIFICACION DE SEGURIDAD
"G1SOPVINH"	M 103.5	BOOL	// G1 LAMPADA SEGURIDAD INACTIVO
"G1MINHIB"	M 103.6	BOOL	// G1 MEMORIA INHIBICION DE SEGURIDAD
"A1MINHIB"	M 104.5	BOOL	// A1 MEMORIA INHIBICION DE SEGURIDAD
"A1SOPVINH"	M 104.6	BOOL	// A1 LAMPADA SEGURIDAD INACTIVO
"A1VINHIB"	M 104.7	BOOL	// A1 VALIDACION DE MODIFICACION DE SEGURIDAD
"A1ACONF"	M 105.0	BOOL	// A1 AUTHORIZACION DE MODIFICACION DE SEGURIDAD
"A2MINHIB"	M 105.2	BOOL	// A2 MEMORIA INHIBICION DE SEGURIDAD
"A2SOPVINH"	M 105.3	BOOL	// A2 LAMPADA SEGURIDAD INACTIVO
"A2VINHIB"	M 105.4	BOOL	// A2 VALIDACION DE MODIFICACION DE SEGURIDAD
"A2ACONF"	M 105.5	BOOL	// A2 AUTHORIZACION DE MODIFICACION DE SEGURIDAD
"D1MINHIB"	M 105.6	BOOL	// D1 MEMORIA INHIBICION DE SEGURIDAD
"D1SOPVINH"	M 105.7	BOOL	// D1 LAMPADA SEGURIDAD INACTIVO
"D1VINHIB"	M 106.0	BOOL	// D1 VALIDACION DE MODIFICACION DE SEGURIDAD
"D1ACONF"	M 106.1	BOOL	// D1 AUTHORIZACION DE MODIFICACION DE SEGURIDAD
"D2MINHIB"	M 106.2	BOOL	// D2 MEMORIA INHIBICION DE SEGURIDAD
"D2SOPVINH"	M 106.3	BOOL	// D2 LAMPADA SEGURIDAD INACTIVO
"D2VINHIB"	M 106.4	BOOL	// D2 VALIDACION DE MODIFICACION DE SEGURIDAD
"D2ACONF"	M 106.5	BOOL	// D2 AUTHORIZACION DE MODIFICACION DE SEGURIDAD
"F1MINHIB"	M 106.6	BOOL	// F1 MEMORIA INHIBICION DE SEGURIDAD
"F1SOPVINH"	M 106.7	BOOL	// F1 LAMPADA SEGURIDAD INACTIVO
"F1VINHIB"	M 107.0	BOOL	// F1 VALIDACION DE MODIFICACION DE SEGURIDAD
"F1ACONF"	M 107.1	BOOL	// F1 AUTHORIZACION DE MODIFICACION DE SEGURIDAD
"F2MINHIB"	M 107.2	BOOL	// F2 MEMORIA INHIBICION DE SEGURIDAD
"F2SOPVINH"	M 107.3	BOOL	// F2 LAMPADA SEGURIDAD INACTIVO
"F2VINHIB"	M 107.4	BOOL	// F2 VALIDACION DE MODIFICACION DE SEGURIDAD
"F2ACONF"	M 107.5	BOOL	// F2 AUTHORIZACION DE MODIFICACION DE SEGURIDAD
"BVLHMI"	M 115.0	BOOL	// Boton validacion lanzamiento de HMI
"AuxActVAL"	M 115.1	BOOL	// Auxiliar activacion boton de validacion
"HBHMI"	M 115.2	BOOL	// Habilitacion boton de validacion
"MAUX_P1M6"	M 150.0	BOOL	// MEMORIA AUXILIAR PISTOLA 1 M6
"MAUX_P2M6"	M 150.1	BOOL	// MEMORIA AUXILIAR PISTOLA 2 M6
"IIT_F0_MGEST_FLUX"	M 200.0	BOOL
"IIT_J0_MGEST_FLUX"	M 200.1	BOOL
"A0_AT_A1"	M 201.0	BOOL	// A0: OPERATOR A1 WORK AUTORIZATION / AUTORISATION DE TRAVAIL OPERATEUR A1
"A0_ET_A1"	M 201.1	BOOL	// A0: OPERATOR A1 WORK COMPLETION / ENREGISTREMENT DE TRAVAIL OPERATEUR A1
"A0_AT_A2"	M 202.0	BOOL	// A0: OPERATOR A2 WORK AUTORIZATION / AUTORISATION DE TRAVAIL OPERATEUR A2
"A0_ET_A2"	M 202.1	BOOL	// A0: OPERATOR A2 WORK COMPLETION / ENREGISTREMENT DE TRAVAIL OPERATEUR A2
"A0_AT_A3"	M 203.0	BOOL	// A0: OPERATOR A3 WORK AUTORIZATION / AUTORISATION DE TRAVAIL OPERATEUR A3
"A0_ET_A3"	M 203.1	BOOL	// A0: OPERATOR A3 WORK COMPLETION / ENREGISTREMENT DE TRAVAIL OPERATEUR A3
"B0_AT_B1"	M 205.0	BOOL	// B0: OPERATOR B1 WORK AUTORIZATION / AUTORISATION DE TRAVAIL OPERATEUR B1
"B0_ET_B1"	M 205.1	BOOL	// B0: OPERATOR B1 WORK COMPLETION / ENREGISTREMENT DE TRAVAIL OPERATEUR B1
"B0_AT_B2"	M 206.0	BOOL	// B0: OPERATOR B2 WORK AUTORIZATION / AUTORISATION DE TRAVAIL OPERATEUR B2
"B0_ET_B2"	M 206.1	BOOL	// B0: OPERATOR B2 WORK COMPLETION / ENREGISTREMENT DE TRAVAIL OPERATEUR B2
"B0_AT_B3"	M 207.0	BOOL	// B0: OPERATOR B3 WORK AUTORIZATION / AUTORISATION DE TRAVAIL OPERATEUR B3
"B0_ET_B3"	M 207.1	BOOL	// B0: OPERATOR B3 WORK COMPLETION / ENREGISTREMENT DE TRAVAIL OPERATEUR B3
"C0_AT_C1"	M 209.0	BOOL	// C0: OPERATOR A1 WORK AUTORIZATION / AUTORISATION DE TRAVAIL OPERATEUR A1
"C0_ET_C1"	M 209.1	BOOL	// C0: OPERATOR A1 WORK COMPLETION / ENREGISTREMENT DE TRAVAIL OPERATEUR A1
"C0_AT_C2"	M 210.0	BOOL	// C0: OPERATOR A2 WORK AUTORIZATION / AUTORISATION DE TRAVAIL OPERATEUR A2
"C0_ET_C2"	M 210.1	BOOL	// C0: OPERATOR A2 WORK COMPLETION / ENREGISTREMENT DE TRAVAIL OPERATEUR A2
"D0_AT_D1"	M 211.0	BOOL	// D0: OPERATOR D1 WORK AUTORIZATION / AUTORISATION DE TRAVAIL OPERATEUR D1
"D0_ET_D1"	M 211.1	BOOL	// D0: OPERATOR D1 WORK COMPLETION / ENREGISTREMENT DE TRAVAIL OPERATEUR D1
"D0_AT_D2"	M 212.0	BOOL	// D0: OPERATOR D2 WORK AUTORIZATION / AUTORISATION DE TRAVAIL OPERATEUR D2
"D0_ET_D2"	M 212.1	BOOL	// D0: OPERATOR D2 WORK COMPLETION / ENREGISTREMENT DE TRAVAIL OPERATEUR D2
"D0_AT_D3"	M 213.0	BOOL	// D0: OPERATOR D3 WORK AUTORIZATION / AUTORISATION DE TRAVAIL OPERATEUR D3
"D0_ET_D3"	M 213.1	BOOL	// D0: OPERATOR D3 WORK COMPLETION / ENREGISTREMENT DE TRAVAIL OPERATEUR D3
"D0_AT_D4"	M 214.0	BOOL	// D0: OPERATOR D4 WORK AUTORIZATION / AUTORISATION DE TRAVAIL OPERATEUR D4
"D0_ET_D4"	M 214.1	BOOL	// D0: OPERATOR D4 WORK COMPLETION / ENREGISTREMENT DE TRAVAIL OPERATEUR D4
"E0_AT_E1"	M 215.0	BOOL	// E0: OPERATOR E1 WORK AUTORIZATION / AUTORISATION DE TRAVAIL OPERATEUR E1
"E0_ET_E1"	M 215.1	BOOL	// E0: OPERATOR E1 WORK COMPLETION / ENREGISTREMENT DE TRAVAIL OPERATEUR E1
"E0_AT_E2"	M 216.0	BOOL	// E0: OPERATOR E2 WORK AUTORIZATION / AUTORISATION DE TRAVAIL OPERATEUR E2
"E0_ET_E2"	M 216.1	BOOL	// E0: OPERATOR E2 WORK COMPLETION / ENREGISTREMENT DE TRAVAIL OPERATEUR E2
"F0_AT_F1"	M 218.0	BOOL	// F0: OPERATOR F1 WORK AUTORIZATION / AUTORISATION DE TRAVAIL OPERATEUR F1
"F0_ET_F1"	M 218.1	BOOL	// F0: OPERATOR F1 WORK COMPLETION / ENREGISTREMENT DE TRAVAIL OPERATEUR F1
"F0_AT_F2"	M 219.0	BOOL	// F0: OPERATOR F2 WORK AUTORIZATION / AUTORISATION DE TRAVAIL OPERATEUR F2
"F0_ET_F2"	M 219.1	BOOL	// F0: OPERATOR F2 WORK COMPLETION / ENREGISTREMENT DE TRAVAIL OPERATEUR F2
"F0_AT_F3"	M 220.0	BOOL	// F0: OPERATOR F3 WORK AUTORIZATION / AUTORISATION DE TRAVAIL OPERATEUR F3
"F0_ET_F3"	M 220.1	BOOL	// F0: OPERATOR F3 WORK COMPLETION / ENREGISTREMENT DE TRAVAIL OPERATEUR F3
"Y0_AT_Y1"	M 221.6	BOOL	// Y0: OPERATOR Y1 WORK AUTORIZATION / AUTORISATION DE TRAVAIL OPERATEUR Y1
"Y0_ET_Y1"	M 221.7	BOOL	// Y0: OPERATOR Y1 WORK COMPLETION / ENREGISTREMENT DE TRAVAIL OPERATEUR Y1
"G0_AT_G1"	M 222.0	BOOL	// G0: OPERATOR G1 WORK AUTORIZATION / AUTORISATION DE TRAVAIL OPERATEUR G1
"G0_ET_G1"	M 222.1	BOOL	// G0: OPERATOR G1 WORK COMPLETION / ENREGISTREMENT DE TRAVAIL OPERATEUR G1
"Z2MANU"	M 222.2	BOOL
"Z2E0_MANUJOG"	M 222.3	BOOL
"G0_AT_G2"	M 223.0	BOOL	// G0: OPERATOR G2 WORK AUTORIZATION / AUTORISATION DE TRAVAIL OPERATEUR G2
"G0_ET_G2"	M 223.1	BOOL	// G0: OPERATOR G2 WORK COMPLETION / ENREGISTREMENT DE TRAVAIL OPERATEUR G2
"K0_AT_K1"	M 227.0	BOOL	// K0: OPERATOR K1 WORK AUTORIZATION / AUTORISATION DE TRAVAIL OPERATEUR K1
"K0_ET_K1"	M 227.1	BOOL	// K0: OPERATOR K1 WORK COMPLETION / ENREGISTREMENT DE TRAVAIL OPERATEUR K1
"L0_AT_L1"	M 230.0	BOOL	// A0: OPERATOR A1 WORK AUTORIZATION / AUTORISATION DE TRAVAIL OPERATEUR A1
"L0_AT_L2"	M 230.1	BOOL	// A0: OPERATOR A2 WORK AUTORIZATION / AUTORISATION DE TRAVAIL OPERATEUR A2
"L0_ET_L1"	M 230.2	BOOL	// A0: OPERATOR A1 WORK COMPLETION / ENREGISTREMENT DE TRAVAIL OPERATEUR A1
"L0_ET_L2"	M 230.3	BOOL	// A0: OPERATOR A2 WORK COMPLETION / ENREGISTREMENT DE TRAVAIL OPERATEUR A2
"M0_AT_M1"	M 230.4	BOOL	// A0: OPERATOR A1 WORK AUTORIZATION / AUTORISATION DE TRAVAIL OPERATEUR A1
"M0_AT_M2"	M 230.5	BOOL	// A0: OPERATOR A2 WORK AUTORIZATION / AUTORISATION DE TRAVAIL OPERATEUR A2
"M0_ET_M1"	M 230.6	BOOL	// A0: OPERATOR A1 WORK COMPLETION / ENREGISTREMENT DE TRAVAIL OPERATEUR A1
"M0_ET_M2"	M 230.7	BOOL	// A0: OPERATOR A2 WORK COMPLETION / ENREGISTREMENT DE TRAVAIL OPERATEUR A2
"N0_AT_N1"	M 231.0	BOOL	// N0: OPERATOR N1 WORK AUTORIZATION / AUTORISATION DE TRAVAIL OPERATEUR N1
"N0_AT_N2"	M 231.1	BOOL	// N0: OPERATOR N2 WORK AUTORIZATION / AUTORISATION DE TRAVAIL OPERATEUR N2
"N0_ET_N1"	M 231.2	BOOL	// N0: OPERATOR N1 WORK COMPLETION / ENREGISTREMENT DE TRAVAIL OPERATEUR N1
"N0_ET_N2"	M 231.3	BOOL	// N0: OPERATOR N2 WORK COMPLETION / ENREGISTREMENT DE TRAVAIL OPERATEUR N2
"MAUXCC1"	M 300.0	BOOL	// Memória Auxiliar Contador Cabeçote 1
"MAUXCC2"	M 300.1	BOOL	// Memória Auxiliar Contador Caabeçote 2
"MAUXCC3"	M 300.2	BOOL	// Memória Auxiliar Contador Cabeçote 3
"MTCT"	M 300.3	BOOL	// Memória Teste Contador Tucker
"CC1_MDEF"	M 300.4	BOOL	// Messagem de Falta de Solda Tucker M5 L52
"CC2_MDEF"	M 300.5	BOOL	// Messagem de Falta de Solda Tucker M6 L52
"CC3_MDEF"	M 300.6	BOOL	// Messagem de Falta de Solda Tucker M5 B52
"CC4_MDEF"	M 300.7	BOOL	// Messagem de Falta de Solda Tucker M6 B52
"CC5_MDEF"	M 301.0	BOOL	// Messagem de Falta de Solda Tucker M5 B52C
"CC6_MDEF"	M 301.1	BOOL	// Messagem de Falta de Solda Tucker M6 B52C
"Y1CRSY0"	M 306.1	BOOL	// Y1: SAFETY RESET CONDITION / CONDITION DE REARMEMENT SECURITE
"SIN_POKA"	M 310.0	BOOL	// SIN POKA YOKE LASER 2 ASIENTOS / 5 ASIENTOS
"SCADA"	M 333.0	BOOL
"MAUX_CT_01"	M 400.0	BOOL	// Memória auxiliar contador M_01
"MAUX_CT_02"	M 400.1	BOOL	// Memória auxiliar contador M6_02
"MBPT"	M 400.2	BOOL	// Memória by pass tucker
"DFT"	M 400.3	BOOL	// Defeito falta de tucker M6
"BP_BIM_A0_X1"	M 500.0	BOOL	// AUXILIAR BY PASS  BIMANUAL - A2
"BP_BIM_B0"	M 500.1	BOOL	// AUXILIAR BY PASS  BIMANUAL B0
"BP_BIM_D0_X1"	M 500.2	BOOL	// AUXILIAR BY PASS  BIMANUAL D2
"BP_BIM_E0"	M 500.3	BOOL	// AUXILIAR BY PASS  BIMANUAL E0
"BP_BIM_F0"	M 500.4	BOOL	// AUXILIAR BY PASS  BIMANUAL F0
"BP_BIM_G0"	M 500.5	BOOL	// AUXILIAR BY PASS  BIMANUAL G0
"BP_BIM_A0_X2"	M 500.7	BOOL	// AUXILIAR BY PASS  BIMANUAL - A2 AND A3
"BP_BIM_D0_X2"	M 501.0	BOOL	// AUXILIAR BY PASS  BIMANUAL D2 - D3 - D4
"BP_BIM_F0_X1"	M 501.2	BOOL	// AUXILIAR BY PASS  BIMANUAL - F2
"BP_BIM_F0_X2"	M 501.3	BOOL	// AUXILIAR BY PASS  BIMANUAL - F2 AND F3
"L1VINHIB"	M 502.0	BOOL
"L1ACONF"	M 502.1	BOOL
"L1MINHIB"	M 502.2	BOOL
"L1DINHIB1"	M 502.3	BOOL
"L2VINHIB"	M 502.4	BOOL
"L2ACONF"	M 502.5	BOOL
"L2MINHIB"	M 502.6	BOOL
"L2DINHIB1"	M 502.7	BOOL
"M1VINHIB"	M 503.0	BOOL
"M1ACONF"	M 503.1	BOOL
"M1MINHIB"	M 503.2	BOOL
"M1DINHIB1"	M 503.3	BOOL
"M2VINHIB"	M 503.4	BOOL
"M2ACONF"	M 503.5	BOOL
"M2MINHIB"	M 503.6	BOOL
"M2DINHIB1"	M 503.7	BOOL
"AUX_AT1_C1_AIO"	M 553.0	BOOL	// AUXILIAR AUTORIZACION DE TRABAJO 1 OPERADOR 1 AIO
"AUX_AT1_C2_AIO"	M 553.1	BOOL	// AUXILIAR AUTORIZACION DE TRABAJO 1 OPERADOR 1 AIO
"AUX_AT1_E1_AIO"	M 553.2	BOOL	// AUXILIAR AUTORIZACION DE TRABAJO 1 OPERADOR 1 AIO
"AUX_AT1_E2_AIO"	M 553.3	BOOL	// AUXILIAR AUTORIZACION DE TRABAJO 1 OPERADOR 2 AIO
"AUX_AT1_G1_AIO"	M 553.4	BOOL	// AUXILIAR AUTORIZACION DE TRABAJO 1 OPERADOR 1 AIO
"AUX_AT1_G2_AIO"	M 553.5	BOOL	// AUXILIAR AUTORIZACION DE TRABAJO 1 OPERADOR 2 AIO
"AUX_AT1_A2_AIO"	M 555.0	BOOL	// AUXILIAR AUTORIZACION DE TRABAJO 1 OPERADOR 2 AIO
"AUX_AT1_A1_AIO"	M 555.1	BOOL	// AUXILIAR AUTORIZACION DE TRABAJO 1 OPERADOR 1 AIO
"AUX_AT1_D1_AIO"	M 555.2	BOOL	// AUXILIAR AUTORIZACION DE TRABAJO 1 OPERADOR 1 AIO
"AUX_AT1_D2_AIO"	M 555.3	BOOL	// AUXILIAR AUTORIZACION DE TRABAJO 1 OPERADOR 2 AIO
"AUX_AT1_F1_AIO"	M 555.4	BOOL	// AUXILIAR AUTORIZACION DE TRABAJO 1 OPERADOR 1 AIO
"AUX_AT1_F2_AIO"	M 555.5	BOOL	// AUXILIAR AUTORIZACION DE TRABAJO 1 OPERADOR 2 AIO
"AUX_AT1_K1_AIO"	M 555.6	BOOL	// AUXILIAR AUTORIZACION DE TRABAJO 1 OPERADOR 1 AIO
"AUX_AT1_B1_AIO"	M 555.7	BOOL	// AUXILIAR AUTORIZACION DE TRABAJO 1 OPERADOR 2 AIO
"MCTRLZA"	M 600.0	BOOL	// MEMORIA CONTROLE ZONA A
"MCTRLZB"	M 600.1	BOOL	// MEMORIA CONTROLE ZONA B
"DPVA"	M 666.0	BOOL
"DPVR"	M 666.1	BOOL
"F_AR_X0VAR"	M 801.0	BOOL	// INFO FALTA CONDIÇAO COM REARME RLV
"F_AR_Y0VAR"	M 801.1	BOOL	// INFO FALTA CONDIÇAO COM REARME RLV
"Y0SOP"	M 802.1	BOOL
"TEST_PGF_Y"	M 870.2	BOOL
"F0BPFL"	M 870.3	BOOL	// F0: BYPASS FLUJO
"J0BPFL"	M 870.4	BOOL	// J0: BYPASS FLUJO
"BSMA"	M 990.1	BOOL	// BIT MODO APRENDIZADO
"MODDEVZ1"	M 992.3	BOOL	// MODO DEVERMINAGE ZONA 1
"MODDEVZ2"	M 992.4	BOOL	// MODO DEVERMINAGE ZONA 2
"Z2SDAPP"	M 992.5	BOOL
"C1CRSC0"	M 992.6	BOOL	// C1: SAFETY RESET CONDITION / CONDITION DE REARMEMENT SECURITE
"C2CRSC0"	M 992.7	BOOL	// C2: SAFETY RESET CONDITION / CONDITION DE REARMEMENT SECURITE
"Y0BPAU"	M 993.1	BOOL
"Y1BPAI"	M 993.3	BOOL
"Z8ESBP"	M 993.4	BOOL
"MODDEVZ3"	M 994.0	BOOL	// MODO DEVERMINAGE ZONA 3
"A0BTPPAD"	M 1010.3	BOOL	// A0 BOTÃO IHM PEÇA PADRÃO
"B0BTPPAD"	M 1010.4	BOOL	// B0 BOTÃO IHM PEÇA PADRÃO
"C0BTPPAD"	M 1010.5	BOOL	// C0 BOTÃO IHM PEÇA PADRÃO
"D0BTPPAD"	M 1010.6	BOOL	// D0 BOTÃO IHM PEÇA PADRÃO
"E0BTPPAD"	M 1011.3	BOOL	// E0 BOTÃO IHM PEÇA PADRÃO
"F0BTPPAD"	M 1011.4	BOOL	// F0 BOTÃO IHM PEÇA PADRÃO
"G0BTPPAD"	M 1011.5	BOOL	// G0 BOTÃO IHM PEÇA PADRÃO
"K0BTPPAD"	M 1012.3	BOOL	// K0 BOTÃO IHM PEÇA PADRÃO
"M_D0FT2DPP"	M 1101.0	BOOL	// Memoria de forzado poke yoke 2
"CMR_H60_TEMP"	M 1106.2	BOOL
"BYPK"	M 1200.0	BOOL	// BYPASS POKAYOKE
"NUEVA DIVERSIDAD"	M 1850.0	BOOL
"CTM_P1M6"	MW 152	WORD	// CONTAGEM PISTOLA 1 M6
"CTM_P2M6"	MW 154	WORD	// CONTAGEM PISTOLA2 M6
"CTM_P1-P2M6"	MW 156	WORD	// CONTAGEM PISTOLA 1 M6 E PISTOLA 2 M6
"B0NORDRE"	MW 300	WORD
"B0wNORDRE"	MW 302	WORD
"C0NORDRE"	MW 304	WORD
"C0wNORDRE"	MW 306	WORD
"E0NORDRE"	MW 308	WORD
"E0wNORDRE"	MW 310	WORD
"G0NORDRE"	MW 312	WORD
"G0wNORDRE"	MW 314	WORD
"J0NORDRE"	MW 316	WORD
"CCT_1"	MW 350	WORD	// Contador Cabeçote Tucker 1
"CCT_2"	MW 352	WORD	// Contador Cabeçote Tucker 2
"SC_CC1-2"	MW 354	WORD	// Resultado Soma Contagem Cabeçote 1e 2
"CCT_3"	MW 356	WORD	// Contador Cabeçote Tucker 3
"SC_CC1-2-3"	MW 358	WORD
"MAUX_BUF_M6_01"	MW 402	WORD	// Memória auxiliar para buffer contador M6_01
"MAUX_BUF_M6_02"	MW 404	WORD	// Memória auxiliar buffer contador M6_02
"MAUX_RS_M6"	MW 406	WORD	// Memória auxiliar soma dos contadores
"CYCL_EXC"	OB 1	OB 1	// EXECUTION CYCLE
"CYC_INT2"	OB 32	OB 32	// CYCLIC INTERRUPT 2
"CYC_INT4"	OB 34	OB 34	// CYCLIC INTERRUPT 4
"I/O_FLT1"	OB 82	OB 82	// I/O POINT FAULT 1
"I/O_FLT2"	OB 83	OB 83	// I/O POINT FAULT 2
"OBNL_FLT"	OB 85	OB 85	// OB NOT LOADED FAULT
"RACK_FLT"	OB 86	OB 86	// LOSS OF RACK FAULT
"COMPLETE RESTART"	OB 100	OB 100	// COMPLETE RESTART
"PROG_ERR"	OB 121	OB 121	// Programming Error
"MOD_ERR"	OB 122	OB 122	// MODULE ACCESS ERROR
"VADI"	Q 0.0	BOOL	// [MOP-IM.M07]: ZONE FAILURE LAMP
"Z1VMCY"	Q 0.1	BOOL	// [MOP-IM.M07]: CYCLE START LAMP
"MOP-IM_M07-08_R1"	Q 0.2	BOOL	// [MOP-IM.M07]: RESERVA
"VAOP"	Q 0.3	BOOL	// [MOP-IM.M07]: OPERATOR REQUEST LAMP
"MOP-IM_M08_R1"	Q 1.0	BOOL	// [MOP-IM.M08]: RESERVA
"MOP-IM_M08_R2"	Q 1.1	BOOL	// [MOP-IM.M08]: RESERVA
"MOP-IM_M08_R3"	Q 1.2	BOOL	// [MOP-IM.M08]: RESERVA
"MOP-IM_M08_R4"	Q 1.3	BOOL	// [MOP-IM.M08]: RESERVA
"Alas"	Q 2.0	BOOL	// [MOP-IM.M09]: RESERVA
"AlaL"	Q 2.1	BOOL	// Alarma Luminosa
"MOP-IM_M09_R3"	Q 2.2	BOOL	// [MOP-IM.M09]: RESERVA
"MOP-IM_M09_R4"	Q 2.3	BOOL	// [MOP-IM.M09]: RESERVA
"Z1VMCY1"	Q 10.0	BOOL	// [Z1ZB.M04]: CYCLE START LAMP
"Z1ZB_M04_R2"	Q 10.1	BOOL	// [Z1ZB.M04]: RESERVA
"Z1ZB_M04_R3"	Q 10.2	BOOL	// [Z1ZB.M04]: RESERVA
"Z1ZB_M04_R4"	Q 10.3	BOOL	// [Z1ZB.M04]: RESERVA
"Z1ZB_M04_R5"	Q 10.4	BOOL	// [Z1ZB.M04]: RESERVA
"Z1ZB_M04_R6"	Q 10.5	BOOL	// [Z1ZB.M04]: RESERVA
"Z1ZB_M04_R7"	Q 10.6	BOOL	// [Z1ZB.M04]: RESERVA
"Z1RCM"	Q 10.7	BOOL	// [Z1ZB.M04]: Z1 GROUND CONTROL RELAY
"Z1RFRO1"	Q 18.0	BOOL	// [Z1ZB.M07]: SAFETY COMMON 1 (RESERVA)
"Z1RFRO2"	Q 18.1	BOOL	// [Z1ZB.M07]: SAFETY COMMON 2 (Z1ES)
"Z1ZB_M07_R1"	Q 18.2	BOOL	// [Z1ZB.M07]: RESERVA
"Z1EV7b"	Q 18.3	BOOL	// [Z1ZB.M07]: Z1 EV 7 bar
"Z2VMCY"	Q 30.0	BOOL	// [Z2ZB.M04]:CYCLE START LAMP
"Z2ZB_M04_R2"	Q 30.1	BOOL	// [Z2ZB.M04]: RESERVA
"Z2ZB_M04_R3"	Q 30.2	BOOL	// [Z2ZB.M04]: RESERVA
"Z2ZB_M04_R4"	Q 30.3	BOOL	// [Z2ZB.M04]: RESERVA
"Z2ZB_M04_R5"	Q 30.4	BOOL	// [Z2ZB.M04]: RESERVA
"Z2ZB_M04_R6"	Q 30.5	BOOL	// [Z2ZB.M04]: RESERVA
"Z2ZB_M04_R7"	Q 30.6	BOOL	// [Z2ZB.M04]: RESERVA
"Z3VMCY"	Q 33.0	BOOL	// (Z2ZB.M05): VOYANT MARCHE CYCLE
"Z3RCM"	Q 33.7	BOOL	// (Z2ZB.M05): RELAIS DE CONTROLE DE MASSE
